LIN {X 0,Y 292.281,Z 425.223,A -85,B 0,C 180,E1 -16748.644,E2 -16748.644} C_VEL
LIN {X 0,Y 292.975,Z 416.538,A -85,B 0,C 180,E1 -16751.064,E2 -16751.064} C_VEL
LIN {X 0,Y 293.77,Z 407.489,A -85,B 0,C 180,E1 -16753.137,E2 -16753.137} C_VEL
LIN {X 0,Y 294.563,Z 398.532,A -85,B 0,C 180,E1 -16754.862,E2 -16754.862} C_VEL
LIN {X 0,Y 295.725,Z 386.736,A -85,B 0,C 180,E1 -16756.748,E2 -16756.748} C_VEL
LIN {X 0,Y 296.927,Z 373.912,A -85,B 0,C 180,E1 -16758.428,E2 -16758.428} C_VEL
LIN {X 0,Y 298.037,Z 360.895,A -85,B 0,C 180,E1 -16759.815,E2 -16759.815} C_VEL
LIN {X 0,Y 298.377,Z 356.314,A -85,B 0,C 180,E1 -16760.24,E2 -16760.24} C_VEL
LIN {X 0,Y 295.222,Z 342.197,A -85,B 0,C 180,E1 -16761.551,E2 -16761.551} C_VEL
LIN {X 0,Y 291.582,Z 327.495,A -85,B 0,C 180,E1 -16762.668,E2 -16762.668} C_VEL
LIN {X 0,Y 290.883,Z 324.481,A -85,B 0,C 180,E1 -16762.869,E2 -16762.869} C_VEL
LIN {X 0,Y 290.897,Z 319.996,A -85,B 0,C 180,E1 -16767.325,E2 -16767.325} C_VEL
LIN {X 0,Y 290.942,Z 316.936,A -85,B 0,C 180,E1 -16770.483,E2 -16770.483} C_VEL
LIN {X 0,Y 290.951,Z 314.87,A -85,B 0,C 180,E1 -16772.743,E2 -16772.743} C_VEL
LIN {X 0,Y 291.348,Z 314.866,A -85,B 0,C 180,E1 -16776.658,E2 -16776.658} C_VEL
LIN {X 0,Y 292.204,Z 318.866,A -85,B 0,C 180,E1 -16780.496,E2 -16780.496} C_VEL
LIN {X 0,Y 292.885,Z 322.76,A -85,B 0,C 180,E1 -16784.097,E2 -16784.097} C_VEL
LIN {X 0,Y 293.355,Z 325.959,A -85,B 0,C 180,E1 -16786.943,E2 -16786.943} C_VEL
LIN {X 0,Y 293.486,Z 329.298,A -85,B 0,C 180,E1 -16789.717,E2 -16789.717} C_VEL
LIN {X 0,Y 293.444,Z 333.828,A -85,B 0,C 180,E1 -16793.219,E2 -16793.219} C_VEL
LIN {X 0,Y 293.478,Z 334.871,A -85,B 0,C 180,E1 -16793.943,E2 -16793.943} C_VEL
LIN {X 0,Y 294.987,Z 338.144,A -85,B 0,C 180,E1 -16794.258,E2 -16794.258} C_VEL
LIN {X 0,Y 301.868,Z 352.507,A -85,B 0,C 180,E1 -16795.778,E2 -16795.778} C_VEL
LIN {X 0,Y 307.005,Z 365.674,A -85,B 0,C 180,E1 -16797.218,E2 -16797.218} C_VEL
LIN {X 0,Y 311.165,Z 379.228,A -85,B 0,C 180,E1 -16798.779,E2 -16798.779} C_VEL
LIN {X 0,Y 312.44,Z 384.388,A -85,B 0,C 180,E1 -16799.396,E2 -16799.396} C_VEL
LIN {X 0,Y 310.407,Z 398.606,A -85,B 0,C 180,E1 -16800.684,E2 -16800.684} C_VEL
LIN {X 0,Y 308.12,Z 411.435,A -85,B 0,C 180,E1 -16802.122,E2 -16802.122} C_VEL
LIN {X 0,Y 305.586,Z 423.472,A -85,B 0,C 180,E1 -16803.759,E2 -16803.759} C_VEL
LIN {X 0,Y 303.036,Z 435.042,A -85,B 0,C 180,E1 -16805.691,E2 -16805.691} C_VEL
LIN {X 0,Y 300.575,Z 444.936,A -85,B 0,C 180,E1 -16807.669,E2 -16807.669} C_VEL
LIN {X 0,Y 298.106,Z 454.57,A -85,B 0,C 180,E1 -16810.01,E2 -16810.01} C_VEL
LIN {X 0,Y 296.027,Z 462.55,A -85,B 0,C 180,E1 -16812.38,E2 -16812.38} C_VEL
LIN {X 0,Y 294.274,Z 469.141,A -85,B 0,C 180,E1 -16814.769,E2 -16814.769} C_VEL
LIN {X 0,Y 292.752,Z 475.226,A -85,B 0,C 180,E1 -16817.522,E2 -16817.522} C_VEL
LIN {X 0,Y 291.602,Z 479.925,A -85,B 0,C 180,E1 -16820.287,E2 -16820.287} C_VEL
LIN {X 0,Y 290.787,Z 483.367,A -85,B 0,C 180,E1 -16823.059,E2 -16823.059} C_VEL
LIN {X 0,Y 290.549,Z 485.611,A -85,B 0,C 180,E1 -16825.838,E2 -16825.838} C_VEL
LIN {X 0,Y 290.207,Z 486.77,A -85,B 0,C 180,E1 -16828.612,E2 -16828.612} C_VEL
LIN {X 0,Y 290.206,Z 486.781,A -85,B 0,C 180,E1 -16831.387,E2 -16831.387} C_VEL
LIN {X 0,Y 290.537,Z 485.67,A -85,B 0,C 180,E1 -16834.161,E2 -16834.161} C_VEL
LIN {X 0,Y 290.788,Z 483.475,A -85,B 0,C 180,E1 -16836.941,E2 -16836.941} C_VEL
LIN {X 0,Y 291.6,Z 480.092,A -85,B 0,C 180,E1 -16839.713,E2 -16839.713} C_VEL
LIN {X 0,Y 292.696,Z 475.454,A -85,B 0,C 180,E1 -16842.48,E2 -16842.48} C_VEL
LIN {X 0,Y 294.228,Z 469.42,A -85,B 0,C 180,E1 -16845.233,E2 -16845.233} C_VEL
LIN {X 0,Y 296.21,Z 461.815,A -85,B 0,C 180,E1 -16847.965,E2 -16847.965} C_VEL
LIN {X 0,Y 298.328,Z 453.69,A -85,B 0,C 180,E1 -16850.333,E2 -16850.333} C_VEL
LIN {X 0,Y 300.921,Z 443.864,A -85,B 0,C 180,E1 -16852.666,E2 -16852.666} C_VEL
LIN {X 0,Y 303.325,Z 433.821,A -85,B 0,C 180,E1 -16854.649,E2 -16854.649} C_VEL
LIN {X 0,Y 305.509,Z 423.937,A -85,B 0,C 180,E1 -16856.284,E2 -16856.284} C_VEL
LIN {X 0,Y 308.026,Z 412.234,A -85,B 0,C 180,E1 -16857.887,E2 -16857.887} C_VEL
LIN {X 0,Y 310.294,Z 399.568,A -85,B 0,C 180,E1 -16859.327,E2 -16859.327} C_VEL
LIN {X 0,Y 312.269,Z 386.595,A -85,B 0,C 180,E1 -16860.523,E2 -16860.523} C_VEL
LIN {X 0,Y 312.394,Z 384.092,A -85,B 0,C 180,E1 -16860.756,E2 -16860.756} C_VEL
LIN {X 0,Y 309.143,Z 372.05,A -85,B 0,C 180,E1 -16862.176,E2 -16862.176} C_VEL
LIN {X 0,Y 304.924,Z 359.837,A -85,B 0,C 180,E1 -16863.543,E2 -16863.543} C_VEL
LIN {X 0,Y 299.653,Z 347.585,A -85,B 0,C 180,E1 -16864.877,E2 -16864.877} C_VEL
LIN {X 0,Y 294.712,Z 337.725,A -85,B 0,C 180,E1 -16865.919,E2 -16865.919} C_VEL
LIN {X 0,Y 293.448,Z 334.746,A -85,B 0,C 180,E1 -16866.235,E2 -16866.235} C_VEL
LIN {X 0,Y 293.518,Z 331.711,A -85,B 0,C 180,E1 -16868.502,E2 -16868.502} C_VEL
LIN {X 0,Y 293.456,Z 327.245,A -85,B 0,C 180,E1 -16872.111,E2 -16872.111} C_VEL
LIN {X 0,Y 293.062,Z 323.956,A -85,B 0,C 180,E1 -16874.978,E2 -16874.978} C_VEL
LIN {X 0,Y 292.466,Z 320.438,A -85,B 0,C 180,E1 -16878.153,E2 -16878.153} C_VEL
LIN {X 0,Y 291.873,Z 317.195,A -85,B 0,C 180,E1 -16881.24,E2 -16881.24} C_VEL
LIN {X 0,Y 291.381,Z 314.808,A -85,B 0,C 180,E1 -16883.777,E2 -16883.777} C_VEL
LIN {X 0,Y 291.366,Z 314.817,A -85,B 0,C 180,E1 -16887.95,E2 -16887.95} C_VEL
LIN {X 0,Y 291.343,Z 314.814,A -85,B 0,C 180,E1 -16891.154,E2 -16891.154} C_VEL
LIN {X 0,Y 291.359,Z 314.803,A -85,B 0,C 180,E1 -16894.266,E2 -16894.266} C_VEL
LIN {X 0,Y 291.369,Z 314.804,A -85,B 0,C 180,E1 -16897.298,E2 -16897.298} C_VEL
LIN {X 0,Y 291.458,Z 314.804,A -85,B 0,C 180,E1 -16900.27,E2 -16900.27} C_VEL
LIN {X 0,Y 291.497,Z 314.792,A -85,B 0,C 180,E1 -16904.665,E2 -16904.665} C_VEL
LIN {X 0,Y 291.485,Z 314.795,A -85,B 0,C 180,E1 -16905.318,E2 -16905.318} C_VEL
LIN {X 0,Y 290.843,Z 314.882,A -85,B 0,C 180,E1 -16906.471,E2 -16906.471} C_VEL
LIN {X 0,Y 288.049,Z 315.231,A -85,B 0,C 180,E1 -16908.35,E2 -16908.35} C_VEL
LIN {X 0,Y 285.681,Z 315.524,A -85,B 0,C 180,E1 -16909.876,E2 -16909.876} C_VEL
LIN {X 0,Y 284.681,Z 315.65,A -85,B 0,C 180,E1 -16911.056,E2 -16911.056} C_VEL
LIN {X 0,Y 284.608,Z 315.659,A -85,B 0,C 180,E1 -16911.456,E2 -16911.456} C_VEL
LIN {X 0,Y 284.574,Z 315.639,A -85,B 0,C 180,E1 -16914.331,E2 -16914.331} C_VEL
LIN {X 0,Y 284.855,Z 315.608,A -85,B 0,C 180,E1 -16918.586,E2 -16918.586} C_VEL
LIN {X 0,Y 284.851,Z 315.619,A -85,B 0,C 180,E1 -16921.414,E2 -16921.414} C_VEL
LIN {X 0,Y 284.658,Z 315.643,A -85,B 0,C 180,E1 -16927.091,E2 -16927.091} C_VEL
LIN {X 0,Y 284.514,Z 315.651,A -85,B 0,C 180,E1 -16929.957,E2 -16929.957} C_VEL
LIN {X 0,Y 284.482,Z 315.673,A -85,B 0,C 180,E1 -16934.303,E2 -16934.303} C_VEL
LIN {X 0,Y 284.425,Z 315.661,A -85,B 0,C 180,E1 -16937.248,E2 -16937.248} C_VEL
LIN {X 0,Y 284.376,Z 315.677,A -85,B 0,C 180,E1 -16940.242,E2 -16940.242} C_VEL
LIN {X 0,Y 284.323,Z 315.694,A -85,B 0,C 180,E1 -16943.854,E2 -16943.854} C_VEL
LIN {X 0,Y 284.283,Z 315.69,A -85,B 0,C 180,E1 -16948.016,E2 -16948.016} C_VEL
LIN {X 0,Y 284.284,Z 315.698,A -85,B 0,C 180,E1 -16951.276,E2 -16951.276} C_VEL
LIN {X 0,Y 284.328,Z 315.807,A -85,B 0,C 180,E1 -16952.243,E2 -16952.243} C_VEL
LIN {X 0,Y 285.91,Z 322.892,A -85,B 0,C 180,E1 -16956.153,E2 -16956.153} C_VEL
LIN {X 0,Y 287.665,Z 330.708,A -85,B 0,C 180,E1 -16960.158,E2 -16960.158} C_VEL
LIN {X 0,Y 289.389,Z 338.363,A -85,B 0,C 180,E1 -16963.831,E2 -16963.831} C_VEL
LIN {X 0,Y 291.295,Z 346.482,A -85,B 0,C 180,E1 -16967.504,E2 -16967.504} C_VEL
LIN {X 0,Y 293.304,Z 354.76,A -85,B 0,C 180,E1 -16970.991,E2 -16970.991} C_VEL
LIN {X 0,Y 293.898,Z 358.498,A -85,B 0,C 180,E1 -16971.839,E2 -16971.839} C_VEL
LIN {X 0,Y 293.238,Z 368.802,A -85,B 0,C 180,E1 -16973.867,E2 -16973.867} C_VEL
LIN {X 0,Y 297.903,Z 390.014,A -85,B 0,C 180,E1 -16975.176,E2 -16975.176} C_VEL
LIN {X 0,Y 300.055,Z 405.991,A -85,B 0,C 180,E1 -16976.266,E2 -16976.266} C_VEL
LIN {X 0,Y 301.158,Z 421.763,A -85,B 0,C 180,E1 -16977.538,E2 -16977.538} C_VEL
LIN {X 0,Y 301.521,Z 436.68,A -85,B 0,C 180,E1 -16978.979,E2 -16978.979} C_VEL
LIN {X 0,Y 301.025,Z 442.79,A -85,B 0,C 180,E1 -16979.594,E2 -16979.594} C_VEL
LIN {X 0,Y 298.222,Z 456.827,A -85,B 0,C 180,E1 -16981.112,E2 -16981.112} C_VEL
LIN {X 0,Y 295.429,Z 469.104,A -85,B 0,C 180,E1 -16982.746,E2 -16982.746} C_VEL
LIN {X 0,Y 292.883,Z 479.435,A -85,B 0,C 180,E1 -16984.41,E2 -16984.41} C_VEL
LIN {X 0,Y 290.393,Z 490.022,A -85,B 0,C 180,E1 -16986.464,E2 -16986.464} C_VEL
LIN {X 0,Y 288.224,Z 499.009,A -85,B 0,C 180,E1 -16988.546,E2 -16988.546} C_VEL
LIN {X 0,Y 286.145,Z 507.863,A -85,B 0,C 180,E1 -16991.008,E2 -16991.008} C_VEL
LIN {X 0,Y 284.681,Z 515.263,A -85,B 0,C 180,E1 -16993.507,E2 -16993.507} C_VEL
LIN {X 0,Y 283.458,Z 522.136,A -85,B 0,C 180,E1 -16996.377,E2 -16996.377} C_VEL
LIN {X 0,Y 282.864,Z 527.542,A -85,B 0,C 180,E1 -16999.261,E2 -16999.261} C_VEL
LIN {X 0,Y 282.743,Z 530.67,A -85,B 0,C 180,E1 -17001.423,E2 -17001.423} C_VEL
LIN {X 0,Y 282.906,Z 533.758,A -85,B 0,C 180,E1 -17004.297,E2 -17004.297} C_VEL
LIN {X 0,Y 283.058,Z 535.604,A -85,B 0,C 180,E1 -17007.154,E2 -17007.154} C_VEL
LIN {X 0,Y 283.209,Z 536.24,A -85,B 0,C 180,E1 -17010,E2 -17010} C_VEL
LIN {X 0,Y 283.107,Z 535.603,A -85,B 0,C 180,E1 -17012.846,E2 -17012.846} C_VEL
LIN {X 0,Y 282.92,Z 533.747,A -85,B 0,C 180,E1 -17015.703,E2 -17015.703} C_VEL
LIN {X 0,Y 282.783,Z 530.648,A -85,B 0,C 180,E1 -17018.576,E2 -17018.576} C_VEL
LIN {X 0,Y 282.981,Z 526.261,A -85,B 0,C 180,E1 -17021.46,E2 -17021.46} C_VEL
LIN {X 0,Y 283.73,Z 520.505,A -85,B 0,C 180,E1 -17024.342,E2 -17024.342} C_VEL
LIN {X 0,Y 285.038,Z 513.22,A -85,B 0,C 180,E1 -17027.21,E2 -17027.21} C_VEL
LIN {X 0,Y 286.735,Z 505.442,A -85,B 0,C 180,E1 -17029.696,E2 -17029.696} C_VEL
LIN {X 0,Y 288.901,Z 496.554,A -85,B 0,C 180,E1 -17032.041,E2 -17032.041} C_VEL
LIN {X 0,Y 291.219,Z 486.613,A -85,B 0,C 180,E1 -17034.222,E2 -17034.222} C_VEL
LIN {X 0,Y 292.965,Z 479.467,A -85,B 0,C 180,E1 -17035.583,E2 -17035.583} C_VEL
LIN {X 0,Y 296.814,Z 468.953,A -85,B 0,C 180,E1 -17037.882,E2 -17037.882} C_VEL
LIN {X 0,Y 301.379,Z 457.024,A -85,B 0,C 180,E1 -17040.052,E2 -17040.052} C_VEL
LIN {X 0,Y 306.225,Z 443.816,A -85,B 0,C 180,E1 -17042.055,E2 -17042.055} C_VEL
LIN {X 0,Y 309.774,Z 429.399,A -85,B 0,C 180,E1 -17044.161,E2 -17044.161} C_VEL
LIN {X 0,Y 311.396,Z 419.284,A -85,B 0,C 180,E1 -17045.66,E2 -17045.66} C_VEL
LIN {X 0,Y 312.435,Z 406.673,A -85,B 0,C 180,E1 -17047.71,E2 -17047.71} C_VEL
LIN {X 0,Y 312.742,Z 394.992,A -85,B 0,C 180,E1 -17049.86,E2 -17049.86} C_VEL
LIN {X 0,Y 312.782,Z 389.058,A -85,B 0,C 180,E1 -17051.089,E2 -17051.089} C_VEL
LIN {X 0,Y 312.133,Z 386.452,A -85,B 0,C 180,E1 -17052.01,E2 -17052.01} C_VEL
LIN {X 0,Y 310.091,Z 381.925,A -85,B 0,C 180,E1 -17054.636,E2 -17054.636} C_VEL
LIN {X 0,Y 309.135,Z 379.146,A -85,B 0,C 180,E1 -17056.998,E2 -17056.998} C_VEL
LIN {X 0,Y 308.913,Z 377.902,A -85,B 0,C 180,E1 -17058.718,E2 -17058.718} C_VEL
LIN {X 0,Y 309.154,Z 377.322,A -85,B 0,C 180,E1 -17060.618,E2 -17060.618} C_VEL
LIN {X 0,Y 309.806,Z 377.672,A -85,B 0,C 180,E1 -17062.56,E2 -17062.56} C_VEL
LIN {X 0,Y 310.718,Z 379.097,A -85,B 0,C 180,E1 -17064.516,E2 -17064.516} C_VEL
LIN {X 0,Y 312.001,Z 381.438,A -85,B 0,C 180,E1 -17066.455,E2 -17066.455} C_VEL
LIN {X 0,Y 313.816,Z 385.948,A -85,B 0,C 180,E1 -17068.997,E2 -17068.997} C_VEL
LIN {X 0,Y 315.619,Z 391.802,A -85,B 0,C 180,E1 -17071.451,E2 -17071.451} C_VEL
LIN {X 0,Y 316.372,Z 395.772,A -85,B 0,C 180,E1 -17072.838,E2 -17072.838} C_VEL
LIN {X 0,Y 311.508,Z 407.708,A -85,B 0,C 180,E1 -17074.879,E2 -17074.879} C_VEL
LIN {X 0,Y 306.8,Z 418.029,A -85,B 0,C 180,E1 -17077.081,E2 -17077.081} C_VEL
LIN {X 0,Y 302.738,Z 426.283,A -85,B 0,C 180,E1 -17079.266,E2 -17079.266} C_VEL
LIN {X 0,Y 299.02,Z 432.975,A -85,B 0,C 180,E1 -17081.501,E2 -17081.501} C_VEL
LIN {X 0,Y 295.395,Z 439.029,A -85,B 0,C 180,E1 -17084.121,E2 -17084.121} C_VEL
LIN {X 0,Y 293.012,Z 442.485,A -85,B 0,C 180,E1 -17086.122,E2 -17086.122} C_VEL
LIN {X 0,Y 290.368,Z 445.829,A -85,B 0,C 180,E1 -17088.835,E2 -17088.835} C_VEL
LIN {X 0,Y 289.19,Z 446.951,A -85,B 0,C 180,E1 -17090.206,E2 -17090.206} C_VEL
LIN {X 0,Y 287.411,Z 448.034,A -85,B 0,C 180,E1 -17092.977,E2 -17092.977} C_VEL
LIN {X 0,Y 286.208,Z 447.668,A -85,B 0,C 180,E1 -17095.776,E2 -17095.776} C_VEL
LIN {X 0,Y 285.571,Z 446.967,A -85,B 0,C 180,E1 -17097.179,E2 -17097.179} C_VEL
LIN {X 0,Y 285.274,Z 445.858,A -85,B 0,C 180,E1 -17098.588,E2 -17098.588} C_VEL
LIN {X 0,Y 284.786,Z 444.375,A -85,B 0,C 180,E1 -17100,E2 -17100} C_VEL
LIN {X 0,Y 284.572,Z 441.39,A -85,B 0,C 180,E1 -17102.123,E2 -17102.123} C_VEL
LIN {X 0,Y 284.356,Z 437.471,A -85,B 0,C 180,E1 -17104.252,E2 -17104.252} C_VEL
LIN {X 0,Y 284.781,Z 432.533,A -85,B 0,C 180,E1 -17106.376,E2 -17106.376} C_VEL
LIN {X 0,Y 285.266,Z 425.416,A -85,B 0,C 180,E1 -17108.847,E2 -17108.847} C_VEL
LIN {X 0,Y 285.982,Z 416.448,A -85,B 0,C 180,E1 -17111.338,E2 -17111.338} C_VEL
LIN {X 0,Y 286.82,Z 407.169,A -85,B 0,C 180,E1 -17113.461,E2 -17113.461} C_VEL
LIN {X 0,Y 287.803,Z 395.908,A -85,B 0,C 180,E1 -17115.582,E2 -17115.582} C_VEL
LIN {X 0,Y 289.17,Z 383.463,A -85,B 0,C 180,E1 -17117.504,E2 -17117.504} C_VEL
LIN {X 0,Y 290.389,Z 369.241,A -85,B 0,C 180,E1 -17119.285,E2 -17119.285} C_VEL
LIN {X 0,Y 291.404,Z 357.506,A -85,B 0,C 180,E1 -17120.47,E2 -17120.47} C_VEL
LIN {X 0,Y 288.49,Z 344.156,A -85,B 0,C 180,E1 -17121.754,E2 -17121.754} C_VEL
LIN {X 0,Y 284.743,Z 328.927,A -85,B 0,C 180,E1 -17122.954,E2 -17122.954} C_VEL
LIN {X 0,Y 283.856,Z 325.076,A -85,B 0,C 180,E1 -17123.23,E2 -17123.23} C_VEL
LIN {X 0,Y 283.857,Z 321.34,A -85,B 0,C 180,E1 -17126.959,E2 -17126.959} C_VEL
LIN {X 0,Y 283.927,Z 318.431,A -85,B 0,C 180,E1 -17129.962,E2 -17129.962} C_VEL
LIN {X 0,Y 283.937,Z 315.742,A -85,B 0,C 180,E1 -17132.994,E2 -17132.994} C_VEL
LIN {X 0,Y 284.182,Z 315.865,A -85,B 0,C 180,E1 -17135.47,E2 -17135.47} C_VEL
LIN {X 0,Y 284.889,Z 318.482,A -85,B 0,C 180,E1 -17138.078,E2 -17138.078} C_VEL
LIN {X 0,Y 285.626,Z 322.113,A -85,B 0,C 180,E1 -17141.633,E2 -17141.633} C_VEL
LIN {X 0,Y 286.302,Z 326.199,A -85,B 0,C 180,E1 -17145.388,E2 -17145.388} C_VEL
LIN {X 0,Y 286.676,Z 329.839,A -85,B 0,C 180,E1 -17148.553,E2 -17148.553} C_VEL
LIN {X 0,Y 286.606,Z 335.245,A -85,B 0,C 180,E1 -17152.825,E2 -17152.825} C_VEL
LIN {X 0,Y 286.734,Z 335.84,A -85,B 0,C 180,E1 -17152.967,E2 -17152.967} C_VEL
LIN {X 0,Y 288.261,Z 338.94,A -85,B 0,C 180,E1 -17153.296,E2 -17153.296} C_VEL
LIN {X 0,Y 294.647,Z 351.97,A -85,B 0,C 180,E1 -17154.758,E2 -17154.758} C_VEL
LIN {X 0,Y 299.925,Z 364.933,A -85,B 0,C 180,E1 -17156.242,E2 -17156.242} C_VEL
LIN {X 0,Y 304.193,Z 378.259,A -85,B 0,C 180,E1 -17157.83,E2 -17157.83} C_VEL
LIN {X 0,Y 306.061,Z 385.562,A -85,B 0,C 180,E1 -17158.744,E2 -17158.744} C_VEL
LIN {X 0,Y 305.672,Z 390.296,A -85,B 0,C 180,E1 -17159.176,E2 -17159.176} C_VEL
LIN {X 0,Y 303.514,Z 403.795,A -85,B 0,C 180,E1 -17160.524,E2 -17160.524} C_VEL
LIN {X 0,Y 300.819,Z 417.049,A -85,B 0,C 180,E1 -17162.143,E2 -17162.143} C_VEL
LIN {X 0,Y 298.096,Z 429.254,A -85,B 0,C 180,E1 -17163.99,E2 -17163.99} C_VEL
LIN {X 0,Y 295.348,Z 440.8,A -85,B 0,C 180,E1 -17166.138,E2 -17166.138} C_VEL
LIN {X 0,Y 292.917,Z 449.874,A -85,B 0,C 180,E1 -17168.167,E2 -17168.167} C_VEL
LIN {X 0,Y 290.461,Z 458.624,A -85,B 0,C 180,E1 -17170.523,E2 -17170.523} C_VEL
LIN {X 0,Y 288.429,Z 466.128,A -85,B 0,C 180,E1 -17172.998,E2 -17172.998} C_VEL
LIN {X 0,Y 286.576,Z 472.977,A -85,B 0,C 180,E1 -17175.804,E2 -17175.804} C_VEL
LIN {X 0,Y 285.176,Z 478.35,A -85,B 0,C 180,E1 -17178.629,E2 -17178.629} C_VEL
LIN {X 0,Y 284.114,Z 482.658,A -85,B 0,C 180,E1 -17181.676,E2 -17181.676} C_VEL
LIN {X 0,Y 283.546,Z 485.244,A -85,B 0,C 180,E1 -17184.31,E2 -17184.31} C_VEL
LIN {X 0,Y 283.505,Z 486.218,A -85,B 0,C 180,E1 -17185.735,E2 -17185.735} C_VEL
LIN {X 0,Y 283.149,Z 487.377,A -85,B 0,C 180,E1 -17188.577,E2 -17188.577} C_VEL
LIN {X 0,Y 283.148,Z 487.388,A -85,B 0,C 180,E1 -17191.422,E2 -17191.422} C_VEL
LIN {X 0,Y 283.494,Z 486.277,A -85,B 0,C 180,E1 -17194.265,E2 -17194.265} C_VEL
LIN {X 0,Y 283.774,Z 484.082,A -85,B 0,C 180,E1 -17197.113,E2 -17197.113} C_VEL
LIN {X 0,Y 284.634,Z 480.698,A -85,B 0,C 180,E1 -17199.953,E2 -17199.953} C_VEL
LIN {X 0,Y 285.778,Z 476.062,A -85,B 0,C 180,E1 -17202.787,E2 -17202.787} C_VEL
LIN {X 0,Y 287.381,Z 470.028,A -85,B 0,C 180,E1 -17205.605,E2 -17205.605} C_VEL
LIN {X 0,Y 289.474,Z 462.421,A -85,B 0,C 180,E1 -17208.398,E2 -17208.398} C_VEL
LIN {X 0,Y 291.697,Z 454.293,A -85,B 0,C 180,E1 -17210.816,E2 -17210.816} C_VEL
LIN {X 0,Y 294.402,Z 444.464,A -85,B 0,C 180,E1 -17213.196,E2 -17213.196} C_VEL
LIN {X 0,Y 296.902,Z 434.419,A -85,B 0,C 180,E1 -17215.219,E2 -17215.219} C_VEL
LIN {X 0,Y 299.181,Z 424.533,A -85,B 0,C 180,E1 -17216.884,E2 -17216.884} C_VEL
LIN {X 0,Y 302.054,Z 411.57,A -85,B 0,C 180,E1 -17218.678,E2 -17218.678} C_VEL
LIN {X 0,Y 304.425,Z 398.618,A -85,B 0,C 180,E1 -17220.14,E2 -17220.14} C_VEL
LIN {X 0,Y 306.217,Z 386.977,A -85,B 0,C 180,E1 -17221.213,E2 -17221.213} C_VEL
LIN {X 0,Y 304.343,Z 378.729,A -85,B 0,C 180,E1 -17222.23,E2 -17222.23} C_VEL
LIN {X 0,Y 300.361,Z 366.023,A -85,B 0,C 180,E1 -17223.747,E2 -17223.747} C_VEL
LIN {X 0,Y 295.504,Z 353.884,A -85,B 0,C 180,E1 -17225.153,E2 -17225.153} C_VEL
LIN {X 0,Y 289.995,Z 342.297,A -85,B 0,C 180,E1 -17226.457,E2 -17226.457} C_VEL
LIN {X 0,Y 286.814,Z 336.104,A -85,B 0,C 180,E1 -17227.141,E2 -17227.141} C_VEL
LIN {X 0,Y 286.611,Z 335.375,A -85,B 0,C 180,E1 -17227.225,E2 -17227.225} C_VEL
LIN {X 0,Y 286.641,Z 331.154,A -85,B 0,C 180,E1 -17230.529,E2 -17230.529} C_VEL
LIN {X 0,Y 286.502,Z 327.733,A -85,B 0,C 180,E1 -17233.381,E2 -17233.381} C_VEL
LIN {X 0,Y 285.797,Z 323.189,A -85,B 0,C 180,E1 -17237.538,E2 -17237.538} C_VEL
LIN {X 0,Y 285.323,Z 320.478,A -85,B 0,C 180,E1 -17240.176,E2 -17240.176} C_VEL
LIN {X 0,Y 284.62,Z 316.929,A -85,B 0,C 180,E1 -17243.656,E2 -17243.656} C_VEL
LIN {X 0,Y 284.343,Z 315.694,A -85,B 0,C 180,E1 -17244.999,E2 -17244.999} C_VEL
LIN {X 0,Y 284.285,Z 315.694,A -85,B 0,C 180,E1 -17248.724,E2 -17248.724} C_VEL
LIN {X 0,Y 284.282,Z 315.7,A -85,B 0,C 180,E1 -17251.984,E2 -17251.984} C_VEL
LIN {X 0,Y 284.323,Z 315.695,A -85,B 0,C 180,E1 -17256.145,E2 -17256.145} C_VEL
LIN {X 0,Y 284.376,Z 315.682,A -85,B 0,C 180,E1 -17259.904,E2 -17259.904} C_VEL
LIN {X 0,Y 284.447,Z 315.667,A -85,B 0,C 180,E1 -17264.492,E2 -17264.492} C_VEL
LIN {X 0,Y 284.482,Z 315.651,A -85,B 0,C 180,E1 -17268.601,E2 -17268.601} C_VEL
LIN {X 0,Y 284.608,Z 315.659,A -85,B 0,C 180,E1 -17271.456,E2 -17271.456} C_VEL
LIN {X 0,Y 283.962,Z 315.743,A -85,B 0,C 180,E1 -17272.636,E2 -17272.636} C_VEL
LIN {X 0,Y 281.129,Z 316.101,A -85,B 0,C 180,E1 -17274.558,E2 -17274.558} C_VEL
LIN {X 0,Y 278.749,Z 316.393,A -85,B 0,C 180,E1 -17276.119,E2 -17276.119} C_VEL
LIN {X 0,Y 277.779,Z 316.507,A -85,B 0,C 180,E1 -17277.329,E2 -17277.329} C_VEL
LIN {X 0,Y 277.728,Z 316.504,A -85,B 0,C 180,E1 -17277.738,E2 -17277.738} C_VEL
LIN {X 0,Y 277.872,Z 316.472,A -85,B 0,C 180,E1 -17280,E2 -17280} C_VEL
LIN {X 0,Y 277.685,Z 316.521,A -85,B 0,C 180,E1 -17282.901,E2 -17282.901} C_VEL
LIN {X 0,Y 277.615,Z 316.522,A -85,B 0,C 180,E1 -17287.272,E2 -17287.272} C_VEL
LIN {X 0,Y 277.457,Z 316.527,A -85,B 0,C 180,E1 -17290.213,E2 -17290.213} C_VEL
LIN {X 0,Y 277.435,Z 316.544,A -85,B 0,C 180,E1 -17294.674,E2 -17294.674} C_VEL
LIN {X 0,Y 277.345,Z 316.564,A -85,B 0,C 180,E1 -17299.234,E2 -17299.234} C_VEL
LIN {X 0,Y 277.279,Z 316.573,A -85,B 0,C 180,E1 -17304.152,E2 -17304.152} C_VEL
LIN {X 0,Y 277.269,Z 316.557,A -85,B 0,C 180,E1 -17307.483,E2 -17307.483} C_VEL
LIN {X 0,Y 277.277,Z 316.626,A -85,B 0,C 180,E1 -17311.518,E2 -17311.518} C_VEL
LIN {X 0,Y 278.781,Z 323.501,A -85,B 0,C 180,E1 -17315.438,E2 -17315.438} C_VEL
LIN {X 0,Y 280.611,Z 331.528,A -85,B 0,C 180,E1 -17319.691,E2 -17319.691} C_VEL
LIN {X 0,Y 282.614,Z 340.564,A -85,B 0,C 180,E1 -17324.131,E2 -17324.131} C_VEL
LIN {X 0,Y 284.495,Z 348.537,A -85,B 0,C 180,E1 -17327.825,E2 -17327.825} C_VEL
LIN {X 0,Y 285.12,Z 350.958,A -85,B 0,C 180,E1 -17328.871,E2 -17328.871} C_VEL
LIN {X 0,Y 287.39,Z 359.286,A -85,B 0,C 180,E1 -17331.047,E2 -17331.047} C_VEL
LIN {X 0,Y 287.427,Z 363.003,A -85,B 0,C 180,E1 -17331.858,E2 -17331.858} C_VEL
LIN {X 0,Y 286.926,Z 368.206,A -85,B 0,C 180,E1 -17332.925,E2 -17332.925} C_VEL
LIN {X 0,Y 291.899,Z 390.588,A -85,B 0,C 180,E1 -17334.404,E2 -17334.404} C_VEL
LIN {X 0,Y 293.918,Z 406.526,A -85,B 0,C 180,E1 -17335.54,E2 -17335.54} C_VEL
LIN {X 0,Y 294.815,Z 421.152,A -85,B 0,C 180,E1 -17336.751,E2 -17336.751} C_VEL
LIN {X 0,Y 295.148,Z 436.187,A -85,B 0,C 180,E1 -17338.245,E2 -17338.245} C_VEL
LIN {X 0,Y 294.694,Z 443.103,A -85,B 0,C 180,E1 -17338.983,E2 -17338.983} C_VEL
LIN {X 0,Y 291.968,Z 456.228,A -85,B 0,C 180,E1 -17340.432,E2 -17340.432} C_VEL
LIN {X 0,Y 289.051,Z 468.498,A -85,B 0,C 180,E1 -17342.093,E2 -17342.093} C_VEL
LIN {X 0,Y 286.435,Z 478.83,A -85,B 0,C 180,E1 -17343.791,E2 -17343.791} C_VEL
LIN {X 0,Y 283.798,Z 489.41,A -85,B 0,C 180,E1 -17345.883,E2 -17345.883} C_VEL
LIN {X 0,Y 281.177,Z 499.77,A -85,B 0,C 180,E1 -17348.366,E2 -17348.366} C_VEL
LIN {X 0,Y 279.06,Z 508.386,A -85,B 0,C 180,E1 -17350.889,E2 -17350.889} C_VEL
LIN {X 0,Y 277.394,Z 516.505,A -85,B 0,C 180,E1 -17353.818,E2 -17353.818} C_VEL
LIN {X 0,Y 276.246,Z 522.992,A -85,B 0,C 180,E1 -17356.764,E2 -17356.764} C_VEL
LIN {X 0,Y 275.729,Z 528.036,A -85,B 0,C 180,E1 -17359.722,E2 -17359.722} C_VEL
LIN {X 0,Y 275.701,Z 531.756,A -85,B 0,C 180,E1 -17362.678,E2 -17362.678} C_VEL
LIN {X 0,Y 275.832,Z 533.147,A -85,B 0,C 180,E1 -17364.151,E2 -17364.151} C_VEL
LIN {X 0,Y 275.963,Z 534.993,A -85,B 0,C 180,E1 -17367.081,E2 -17367.081} C_VEL
LIN {X 0,Y 276.093,Z 535.469,A -85,B 0,C 180,E1 -17368.542,E2 -17368.542} C_VEL
LIN {X 0,Y 276.143,Z 535.633,A -85,B 0,C 180,E1 -17370,E2 -17370} C_VEL
LIN {X 0,Y 276.01,Z 534.992,A -85,B 0,C 180,E1 -17372.919,E2 -17372.919} C_VEL
LIN {X 0,Y 275.814,Z 532.68,A -85,B 0,C 180,E1 -17376.407,E2 -17376.407} C_VEL
LIN {X 0,Y 275.72,Z 529.092,A -85,B 0,C 180,E1 -17379.537,E2 -17379.537} C_VEL
LIN {X 0,Y 276.12,Z 524.357,A -85,B 0,C 180,E1 -17382.495,E2 -17382.495} C_VEL
LIN {X 0,Y 277.016,Z 518.322,A -85,B 0,C 180,E1 -17385.405,E2 -17385.405} C_VEL
LIN {X 0,Y 278.566,Z 510.531,A -85,B 0,C 180,E1 -17388.383,E2 -17388.383} C_VEL
LIN {X 0,Y 280.606,Z 502.317,A -85,B 0,C 180,E1 -17390.91,E2 -17390.91} C_VEL
LIN {X 0,Y 283.002,Z 492.465,A -85,B 0,C 180,E1 -17393.412,E2 -17393.412} C_VEL
LIN {X 0,Y 285.548,Z 482.494,A -85,B 0,C 180,E1 -17395.513,E2 -17395.513} C_VEL
LIN {X 0,Y 289.975,Z 471.309,A -85,B 0,C 180,E1 -17398.205,E2 -17398.205} C_VEL
LIN {X 0,Y 295.424,Z 458.079,A -85,B 0,C 180,E1 -17400.763,E2 -17400.763} C_VEL
LIN {X 0,Y 300.415,Z 445.598,A -85,B 0,C 180,E1 -17402.752,E2 -17402.752} C_VEL
LIN {X 0,Y 304.302,Z 431.965,A -85,B 0,C 180,E1 -17404.863,E2 -17404.863} C_VEL
LIN {X 0,Y 306.258,Z 422.529,A -85,B 0,C 180,E1 -17406.353,E2 -17406.353} C_VEL
LIN {X 0,Y 307.74,Z 410.784,A -85,B 0,C 180,E1 -17408.349,E2 -17408.349} C_VEL
LIN {X 0,Y 308.684,Z 398.969,A -85,B 0,C 180,E1 -17410.645,E2 -17410.645} C_VEL
LIN {X 0,Y 308.934,Z 394.037,A -85,B 0,C 180,E1 -17411.714,E2 -17411.714} C_VEL
LIN {X 0,Y 308.68,Z 392.72,A -85,B 0,C 180,E1 -17412.2,E2 -17412.2} C_VEL
LIN {X 0,Y 307.271,Z 389.29,A -85,B 0,C 180,E1 -17414.101,E2 -17414.101} C_VEL
LIN {X 0,Y 306.209,Z 386.119,A -85,B 0,C 180,E1 -17416.485,E2 -17416.485} C_VEL
LIN {X 0,Y 305.812,Z 384.089,A -85,B 0,C 180,E1 -17419.323,E2 -17419.323} C_VEL
LIN {X 0,Y 306.202,Z 383.736,A -85,B 0,C 180,E1 -17421.705,E2 -17421.705} C_VEL
LIN {X 0,Y 306.812,Z 384.516,A -85,B 0,C 180,E1 -17423.447,E2 -17423.447} C_VEL
LIN {X 0,Y 308.086,Z 387.118,A -85,B 0,C 180,E1 -17426.102,E2 -17426.102} C_VEL
LIN {X 0,Y 309.454,Z 391.026,A -85,B 0,C 180,E1 -17428.51,E2 -17428.51} C_VEL
LIN {X 0,Y 310.778,Z 396.356,A -85,B 0,C 180,E1 -17430.964,E2 -17430.964} C_VEL
LIN {X 0,Y 311.134,Z 398.401,A -85,B 0,C 180,E1 -17431.758,E2 -17431.758} C_VEL
LIN {X 0,Y 311.001,Z 400.34,A -85,B 0,C 180,E1 -17432.329,E2 -17432.329} C_VEL
LIN {X 0,Y 306.318,Z 410.593,A -85,B 0,C 180,E1 -17434.156,E2 -17434.156} C_VEL
LIN {X 0,Y 301.513,Z 420.203,A -85,B 0,C 180,E1 -17436.292,E2 -17436.292} C_VEL
LIN {X 0,Y 297.187,Z 428.2,A -85,B 0,C 180,E1 -17438.497,E2 -17438.497} C_VEL
LIN {X 0,Y 292.718,Z 435.594,A -85,B 0,C 180,E1 -17441.087,E2 -17441.087} C_VEL
LIN {X 0,Y 288.902,Z 441.288,A -85,B 0,C 180,E1 -17443.755,E2 -17443.755} C_VEL
LIN {X 0,Y 286.433,Z 444.53,A -85,B 0,C 180,E1 -17445.797,E2 -17445.797} C_VEL
LIN {X 0,Y 283.62,Z 447.558,A -85,B 0,C 180,E1 -17448.566,E2 -17448.566} C_VEL
LIN {X 0,Y 281.369,Z 449.145,A -85,B 0,C 180,E1 -17451.381,E2 -17451.381} C_VEL
LIN {X 0,Y 279.821,Z 449.273,A -85,B 0,C 180,E1 -17454.234,E2 -17454.234} C_VEL
LIN {X 0,Y 279.229,Z 448.814,A -85,B 0,C 180,E1 -17455.67,E2 -17455.67} C_VEL
LIN {X 0,Y 278.566,Z 447.994,A -85,B 0,C 180,E1 -17457.108,E2 -17457.108} C_VEL
LIN {X 0,Y 278.255,Z 446.744,A -85,B 0,C 180,E1 -17458.553,E2 -17458.553} C_VEL
LIN {X 0,Y 277.684,Z 444.229,A -85,B 0,C 180,E1 -17460.725,E2 -17460.725} C_VEL
LIN {X 0,Y 277.381,Z 440.772,A -85,B 0,C 180,E1 -17462.905,E2 -17462.905} C_VEL
LIN {X 0,Y 277.455,Z 436.333,A -85,B 0,C 180,E1 -17465.086,E2 -17465.086} C_VEL
LIN {X 0,Y 277.939,Z 429.861,A -85,B 0,C 180,E1 -17467.629,E2 -17467.629} C_VEL
LIN {X 0,Y 278.537,Z 421.504,A -85,B 0,C 180,E1 -17470.247,E2 -17470.247} C_VEL
LIN {X 0,Y 279.247,Z 413.322,A -85,B 0,C 180,E1 -17472.353,E2 -17472.353} C_VEL
LIN {X 0,Y 280.156,Z 403.167,A -85,B 0,C 180,E1 -17474.529,E2 -17474.529} C_VEL
LIN {X 0,Y 281.43,Z 390.835,A -85,B 0,C 180,E1 -17476.69,E2 -17476.69} C_VEL
LIN {X 0,Y 282.662,Z 378.353,A -85,B 0,C 180,E1 -17478.482,E2 -17478.482} C_VEL
LIN {X 0,Y 283.968,Z 364.057,A -85,B 0,C 180,E1 -17480.15,E2 -17480.15} C_VEL
LIN {X 0,Y 284.374,Z 357.804,A -85,B 0,C 180,E1 -17480.772,E2 -17480.772} C_VEL
LIN {X 0,Y 280.925,Z 342.8,A -85,B 0,C 180,E1 -17482.233,E2 -17482.233} C_VEL
LIN {X 0,Y 277.287,Z 327.78,A -85,B 0,C 180,E1 -17483.41,E2 -17483.41} C_VEL
LIN {X 0,Y 276.821,Z 325.692,A -85,B 0,C 180,E1 -17483.566,E2 -17483.566} C_VEL
LIN {X 0,Y 276.841,Z 321.982,A -85,B 0,C 180,E1 -17487.311,E2 -17487.311} C_VEL
LIN {X 0,Y 276.884,Z 318.925,A -85,B 0,C 180,E1 -17490.508,E2 -17490.508} C_VEL
LIN {X 0,Y 276.894,Z 316.617,A -85,B 0,C 180,E1 -17493.113,E2 -17493.113} C_VEL
LIN {X 0,Y 276.984,Z 316.706,A -85,B 0,C 180,E1 -17493.932,E2 -17493.932} C_VEL
LIN {X 0,Y 277.953,Z 319.947,A -85,B 0,C 180,E1 -17497.361,E2 -17497.361} C_VEL
LIN {X 0,Y 278.721,Z 323.564,A -85,B 0,C 180,E1 -17500.965,E2 -17500.965} C_VEL
LIN {X 0,Y 279.492,Z 328.09,A -85,B 0,C 180,E1 -17505.244,E2 -17505.244} C_VEL
LIN {X 0,Y 279.784,Z 330.398,A -85,B 0,C 180,E1 -17507.295,E2 -17507.295} C_VEL
LIN {X 0,Y 279.835,Z 333.88,A -85,B 0,C 180,E1 -17510.176,E2 -17510.176} C_VEL
LIN {X 0,Y 279.886,Z 336.179,A -85,B 0,C 180,E1 -17511.893,E2 -17511.893} C_VEL
LIN {X 0,Y 281.481,Z 339.551,A -85,B 0,C 180,E1 -17512.26,E2 -17512.26} C_VEL
LIN {X 0,Y 287.749,Z 352.113,A -85,B 0,C 180,E1 -17513.755,E2 -17513.755} C_VEL
LIN {X 0,Y 293.214,Z 365.239,A -85,B 0,C 180,E1 -17515.336,E2 -17515.336} C_VEL
LIN {X 0,Y 297.207,Z 377.357,A -85,B 0,C 180,E1 -17516.832,E2 -17516.832} C_VEL
LIN {X 0,Y 299.98,Z 388.263,A -85,B 0,C 180,E1 -17518.256,E2 -17518.256} C_VEL
LIN {X 0,Y 297.919,Z 401.326,A -85,B 0,C 180,E1 -17519.523,E2 -17519.523} C_VEL
LIN {X 0,Y 295.159,Z 415.141,A -85,B 0,C 180,E1 -17521.172,E2 -17521.172} C_VEL
LIN {X 0,Y 292.498,Z 426.547,A -85,B 0,C 180,E1 -17522.837,E2 -17522.837} C_VEL
LIN {X 0,Y 289.775,Z 437.979,A -85,B 0,C 180,E1 -17524.885,E2 -17524.885} C_VEL
LIN {X 0,Y 287.118,Z 447.601,A -85,B 0,C 180,E1 -17526.943,E2 -17526.943} C_VEL
LIN {X 0,Y 284.46,Z 456.987,A -85,B 0,C 180,E1 -17529.386,E2 -17529.386} C_VEL
LIN {X 0,Y 282.271,Z 464.783,A -85,B 0,C 180,E1 -17531.867,E2 -17531.867} C_VEL
LIN {X 0,Y 280.159,Z 472.031,A -85,B 0,C 180,E1 -17534.728,E2 -17534.728} C_VEL
LIN {X 0,Y 278.595,Z 477.761,A -85,B 0,C 180,E1 -17537.618,E2 -17537.618} C_VEL
LIN {X 0,Y 277.656,Z 481.144,A -85,B 0,C 180,E1 -17539.794,E2 -17539.794} C_VEL
LIN {X 0,Y 276.76,Z 484.583,A -85,B 0,C 180,E1 -17542.705,E2 -17542.705} C_VEL
LIN {X 0,Y 276.462,Z 486.826,A -85,B 0,C 180,E1 -17545.626,E2 -17545.626} C_VEL
LIN {X 0,Y 276.094,Z 487.984,A -85,B 0,C 180,E1 -17548.541,E2 -17548.541} C_VEL
LIN {X 0,Y 276.093,Z 487.995,A -85,B 0,C 180,E1 -17551.458,E2 -17551.458} C_VEL
LIN {X 0,Y 276.451,Z 486.884,A -85,B 0,C 180,E1 -17554.374,E2 -17554.374} C_VEL
LIN {X 0,Y 276.764,Z 484.689,A -85,B 0,C 180,E1 -17557.294,E2 -17557.294} C_VEL
LIN {X 0,Y 277.652,Z 481.307,A -85,B 0,C 180,E1 -17560.206,E2 -17560.206} C_VEL
LIN {X 0,Y 278.873,Z 476.669,A -85,B 0,C 180,E1 -17563.109,E2 -17563.109} C_VEL
LIN {X 0,Y 280.55,Z 470.635,A -85,B 0,C 180,E1 -17565.995,E2 -17565.995} C_VEL
LIN {X 0,Y 282.755,Z 463.026,A -85,B 0,C 180,E1 -17568.851,E2 -17568.851} C_VEL
LIN {X 0,Y 285.1,Z 454.895,A -85,B 0,C 180,E1 -17571.321,E2 -17571.321} C_VEL
LIN {X 0,Y 287.913,Z 445.064,A -85,B 0,C 180,E1 -17573.751,E2 -17573.751} C_VEL
LIN {X 0,Y 290.507,Z 435.018,A -85,B 0,C 180,E1 -17575.814,E2 -17575.814} C_VEL
LIN {X 0,Y 293.182,Z 424.079,A -85,B 0,C 180,E1 -17577.673,E2 -17577.673} C_VEL
LIN {X 0,Y 296.112,Z 410.847,A -85,B 0,C 180,E1 -17579.504,E2 -17579.504} C_VEL
LIN {X 0,Y 298.662,Z 397.598,A -85,B 0,C 180,E1 -17580.981,E2 -17580.981} C_VEL
LIN {X 0,Y 300.04,Z 388.603,A -85,B 0,C 180,E1 -17581.822,E2 -17581.822} C_VEL
LIN {X 0,Y 297.464,Z 377.983,A -85,B 0,C 180,E1 -17583.201,E2 -17583.201} C_VEL
LIN {X 0,Y 293.313,Z 365.35,A -85,B 0,C 180,E1 -17584.769,E2 -17584.769} C_VEL
LIN {X 0,Y 287.9,Z 352.437,A -85,B 0,C 180,E1 -17586.334,E2 -17586.334} C_VEL
LIN {X 0,Y 283.31,Z 343.044,A -85,B 0,C 180,E1 -17587.456,E2 -17587.456} C_VEL
LIN {X 0,Y 280.938,Z 338.728,A -85,B 0,C 180,E1 -17587.985,E2 -17587.985} C_VEL
LIN {X 0,Y 279.845,Z 336.006,A -85,B 0,C 180,E1 -17588.29,E2 -17588.29} C_VEL
LIN {X 0,Y 279.821,Z 332.49,A -85,B 0,C 180,E1 -17591.107,E2 -17591.107} C_VEL
LIN {X 0,Y 279.738,Z 329.952,A -85,B 0,C 180,E1 -17593.232,E2 -17593.232} C_VEL
LIN {X 0,Y 279.075,Z 325.693,A -85,B 0,C 180,E1 -17597.16,E2 -17597.16} C_VEL
LIN {X 0,Y 278.402,Z 321.963,A -85,B 0,C 180,E1 -17600.868,E2 -17600.868} C_VEL
LIN {X 0,Y 277.68,Z 318.371,A -85,B 0,C 180,E1 -17604.4,E2 -17604.4} C_VEL
LIN {X 0,Y 277.236,Z 316.566,A -85,B 0,C 180,E1 -17606.322,E2 -17606.322} C_VEL
LIN {X 0,Y 277.261,Z 316.561,A -85,B 0,C 180,E1 -17609.538,E2 -17609.538} C_VEL
LIN {X 0,Y 277.291,Z 316.56,A -85,B 0,C 180,E1 -17612.857,E2 -17612.857} C_VEL
LIN {X 0,Y 277.284,Z 316.572,A -85,B 0,C 180,E1 -17616.075,E2 -17616.075} C_VEL
LIN {X 0,Y 277.329,Z 316.566,A -85,B 0,C 180,E1 -17620.765,E2 -17620.765} C_VEL
LIN {X 0,Y 277.41,Z 316.554,A -85,B 0,C 180,E1 -17625.324,E2 -17625.324} C_VEL
LIN {X 0,Y 277.457,Z 316.536,A -85,B 0,C 180,E1 -17629.787,E2 -17629.787} C_VEL
LIN {X 0,Y 277.601,Z 316.514,A -85,B 0,C 180,E1 -17632.728,E2 -17632.728} C_VEL
LIN {X 0,Y 277.728,Z 316.504,A -85,B 0,C 180,E1 -17637.738,E2 -17637.738} C_VEL
LIN {X 0,Y 277.126,Z 316.569,A -85,B 0,C 180,E1 -17638.95,E2 -17638.95} C_VEL
LIN {X 0,Y 274.244,Z 316.931,A -85,B 0,C 180,E1 -17640.921,E2 -17640.921} C_VEL
LIN {X 0,Y 271.705,Z 317.266,A -85,B 0,C 180,E1 -17642.523,E2 -17642.523} C_VEL
LIN {X 0,Y 270.549,Z 317.396,A -85,B 0,C 180,E1 -17643.766,E2 -17643.766} C_VEL
LIN {X 0,Y 270.423,Z 317.405,A -85,B 0,C 180,E1 -17644.189,E2 -17644.189} C_VEL
LIN {X 0,Y 270.574,Z 317.401,A -85,B 0,C 180,E1 -17647.462,E2 -17647.462} C_VEL
LIN {X 0,Y 270.41,Z 317.402,A -85,B 0,C 180,E1 -17650.482,E2 -17650.482} C_VEL
LIN {X 0,Y 270.403,Z 317.413,A -85,B 0,C 180,E1 -17655.064,E2 -17655.064} C_VEL
LIN {X 0,Y 270.301,Z 317.437,A -85,B 0,C 180,E1 -17659.755,E2 -17659.755} C_VEL
LIN {X 0,Y 270.224,Z 317.449,A -85,B 0,C 180,E1 -17664.59,E2 -17664.59} C_VEL
LIN {X 0,Y 270.198,Z 317.442,A -85,B 0,C 180,E1 -17667.917,E2 -17667.917} C_VEL
LIN {X 0,Y 270.232,Z 317.635,A -85,B 0,C 180,E1 -17670.881,E2 -17670.881} C_VEL
LIN {X 0,Y 271.688,Z 324.044,A -85,B 0,C 180,E1 -17674.687,E2 -17674.687} C_VEL
LIN {X 0,Y 273.376,Z 331.692,A -85,B 0,C 180,E1 -17678.878,E2 -17678.878} C_VEL
LIN {X 0,Y 275.035,Z 339.202,A -85,B 0,C 180,E1 -17682.731,E2 -17682.731} C_VEL
LIN {X 0,Y 276.801,Z 346.705,A -85,B 0,C 180,E1 -17686.354,E2 -17686.354} C_VEL
LIN {X 0,Y 279.779,Z 357.452,A -85,B 0,C 180,E1 -17689.452,E2 -17689.452} C_VEL
LIN {X 0,Y 281.103,Z 362.432,A -85,B 0,C 180,E1 -17690.809,E2 -17690.809} C_VEL
LIN {X 0,Y 280.721,Z 367.678,A -85,B 0,C 180,E1 -17691.966,E2 -17691.966} C_VEL
LIN {X 0,Y 285.47,Z 388.984,A -85,B 0,C 180,E1 -17693.426,E2 -17693.426} C_VEL
LIN {X 0,Y 287.449,Z 403.824,A -85,B 0,C 180,E1 -17694.506,E2 -17694.506} C_VEL
LIN {X 0,Y 288.494,Z 417.85,A -85,B 0,C 180,E1 -17695.692,E2 -17695.692} C_VEL
LIN {X 0,Y 288.852,Z 432.882,A -85,B 0,C 180,E1 -17697.173,E2 -17697.173} C_VEL
LIN {X 0,Y 288.49,Z 442.758,A -85,B 0,C 180,E1 -17698.271,E2 -17698.271} C_VEL
LIN {X 0,Y 285.72,Z 455.625,A -85,B 0,C 180,E1 -17699.719,E2 -17699.719} C_VEL
LIN {X 0,Y 282.769,Z 467.897,A -85,B 0,C 180,E1 -17701.417,E2 -17701.417} C_VEL
LIN {X 0,Y 280.008,Z 478.223,A -85,B 0,C 180,E1 -17703.142,E2 -17703.142} C_VEL
LIN {X 0,Y 277.229,Z 488.798,A -85,B 0,C 180,E1 -17705.274,E2 -17705.274} C_VEL
LIN {X 0,Y 274.887,Z 497.784,A -85,B 0,C 180,E1 -17707.449,E2 -17707.449} C_VEL
LIN {X 0,Y 272.58,Z 506.634,A -85,B 0,C 180,E1 -17710.024,E2 -17710.024} C_VEL
LIN {X 0,Y 270.855,Z 514.026,A -85,B 0,C 180,E1 -17712.639,E2 -17712.639} C_VEL
LIN {X 0,Y 269.493,Z 520.903,A -85,B 0,C 180,E1 -17715.656,E2 -17715.656} C_VEL
LIN {X 0,Y 268.755,Z 526.309,A -85,B 0,C 180,E1 -17718.69,E2 -17718.69} C_VEL
LIN {X 0,Y 268.587,Z 529.44,A -85,B 0,C 180,E1 -17720.968,E2 -17720.968} C_VEL
LIN {X 0,Y 268.738,Z 532.534,A -85,B 0,C 180,E1 -17723.996,E2 -17723.996} C_VEL
LIN {X 0,Y 268.87,Z 534.382,A -85,B 0,C 180,E1 -17727.004,E2 -17727.004} C_VEL
LIN {X 0,Y 269.029,Z 534.861,A -85,B 0,C 180,E1 -17728.503,E2 -17728.503} C_VEL
LIN {X 0,Y 269.079,Z 535.025,A -85,B 0,C 180,E1 -17730,E2 -17730} C_VEL
LIN {X 0,Y 269.045,Z 534.861,A -85,B 0,C 180,E1 -17731.497,E2 -17731.497} C_VEL
LIN {X 0,Y 268.776,Z 533.599,A -85,B 0,C 180,E1 -17734.5,E2 -17734.5} C_VEL
LIN {X 0,Y 268.73,Z 532.221,A -85,B 0,C 180,E1 -17736.385,E2 -17736.385} C_VEL
LIN {X 0,Y 268.634,Z 528.474,A -85,B 0,C 180,E1 -17739.791,E2 -17739.791} C_VEL
LIN {X 0,Y 269.085,Z 523.737,A -85,B 0,C 180,E1 -17742.827,E2 -17742.827} C_VEL
LIN {X 0,Y 270.155,Z 517.362,A -85,B 0,C 180,E1 -17745.966,E2 -17745.966} C_VEL
LIN {X 0,Y 271.726,Z 509.911,A -85,B 0,C 180,E1 -17748.863,E2 -17748.863} C_VEL
LIN {X 0,Y 273.898,Z 501.7,A -85,B 0,C 180,E1 -17751.448,E2 -17751.448} C_VEL
LIN {X 0,Y 276.402,Z 491.848,A -85,B 0,C 180,E1 -17754.006,E2 -17754.006} C_VEL
LIN {X 0,Y 278.631,Z 484.049,A -85,B 0,C 180,E1 -17755.792,E2 -17755.792} C_VEL
LIN {X 0,Y 283.116,Z 473.445,A -85,B 0,C 180,E1 -17758.546,E2 -17758.546} C_VEL
LIN {X 0,Y 287.923,Z 462.746,A -85,B 0,C 180,E1 -17760.837,E2 -17760.837} C_VEL
LIN {X 0,Y 293.682,Z 449.941,A -85,B 0,C 180,E1 -17763.081,E2 -17763.081} C_VEL
LIN {X 0,Y 297.65,Z 438.689,A -85,B 0,C 180,E1 -17764.931,E2 -17764.931} C_VEL
LIN {X 0,Y 300.864,Z 426.955,A -85,B 0,C 180,E1 -17766.85,E2 -17766.85} C_VEL
LIN {X 0,Y 303.086,Z 414.638,A -85,B 0,C 180,E1 -17769.048,E2 -17769.048} C_VEL
LIN {X 0,Y 304.486,Z 403.636,A -85,B 0,C 180,E1 -17771.278,E2 -17771.278} C_VEL
LIN {X 0,Y 304.855,Z 400.573,A -85,B 0,C 180,E1 -17771.956,E2 -17771.956} C_VEL
LIN {X 0,Y 304.943,Z 398.633,A -85,B 0,C 180,E1 -17772.481,E2 -17772.481} C_VEL
LIN {X 0,Y 303.838,Z 395.554,A -85,B 0,C 180,E1 -17774.188,E2 -17774.188} C_VEL
LIN {X 0,Y 303.031,Z 393.07,A -85,B 0,C 180,E1 -17775.969,E2 -17775.969} C_VEL
LIN {X 0,Y 302.547,Z 391.147,A -85,B 0,C 180,E1 -17778.017,E2 -17778.017} C_VEL
LIN {X 0,Y 302.507,Z 390.09,A -85,B 0,C 180,E1 -17780.057,E2 -17780.057} C_VEL
LIN {X 0,Y 302.841,Z 390.099,A -85,B 0,C 180,E1 -17782.096,E2 -17782.096} C_VEL
LIN {X 0,Y 303.596,Z 391.623,A -85,B 0,C 180,E1 -17784.639,E2 -17784.639} C_VEL
LIN {X 0,Y 304.546,Z 394.367,A -85,B 0,C 180,E1 -17786.945,E2 -17786.945} C_VEL
LIN {X 0,Y 305.394,Z 397.845,A -85,B 0,C 180,E1 -17788.979,E2 -17788.979} C_VEL
LIN {X 0,Y 306.146,Z 402.613,A -85,B 0,C 180,E1 -17791.179,E2 -17791.179} C_VEL
LIN {X 0,Y 306.094,Z 403.55,A -85,B 0,C 180,E1 -17791.511,E2 -17791.511} C_VEL
LIN {X 0,Y 301.386,Z 413.142,A -85,B 0,C 180,E1 -17793.328,E2 -17793.328} C_VEL
LIN {X 0,Y 296.328,Z 422.503,A -85,B 0,C 180,E1 -17795.478,E2 -17795.478} C_VEL
LIN {X 0,Y 292.361,Z 429.202,A -85,B 0,C 180,E1 -17797.38,E2 -17797.38} C_VEL
LIN {X 0,Y 287.509,Z 436.59,A -85,B 0,C 180,E1 -17799.988,E2 -17799.988} C_VEL
LIN {X 0,Y 283.38,Z 442.341,A -85,B 0,C 180,E1 -17802.686,E2 -17802.686} C_VEL
LIN {X 0,Y 279.831,Z 446.531,A -85,B 0,C 180,E1 -17805.454,E2 -17805.454} C_VEL
LIN {X 0,Y 276.883,Z 449.273,A -85,B 0,C 180,E1 -17808.284,E2 -17808.284} C_VEL
LIN {X 0,Y 274.526,Z 450.606,A -85,B 0,C 180,E1 -17811.164,E2 -17811.164} C_VEL
LIN {X 0,Y 272.867,Z 450.518,A -85,B 0,C 180,E1 -17814.087,E2 -17814.087} C_VEL
LIN {X 0,Y 272.248,Z 449.906,A -85,B 0,C 180,E1 -17815.558,E2 -17815.558} C_VEL
LIN {X 0,Y 271.56,Z 448.956,A -85,B 0,C 180,E1 -17817.033,E2 -17817.033} C_VEL
LIN {X 0,Y 271.235,Z 447.606,A -85,B 0,C 180,E1 -17818.515,E2 -17818.515} C_VEL
LIN {X 0,Y 270.644,Z 444.9,A -85,B 0,C 180,E1 -17820.744,E2 -17820.744} C_VEL
LIN {X 0,Y 270.306,Z 441.291,A -85,B 0,C 180,E1 -17822.981,E2 -17822.981} C_VEL
LIN {X 0,Y 270.403,Z 436.715,A -85,B 0,C 180,E1 -17825.219,E2 -17825.219} C_VEL
LIN {X 0,Y 270.888,Z 429.867,A -85,B 0,C 180,E1 -17827.869,E2 -17827.869} C_VEL
LIN {X 0,Y 271.518,Z 421.653,A -85,B 0,C 180,E1 -17830.439,E2 -17830.439} C_VEL
LIN {X 0,Y 272.275,Z 412.997,A -85,B 0,C 180,E1 -17832.674,E2 -17832.674} C_VEL
LIN {X 0,Y 273.247,Z 402.578,A -85,B 0,C 180,E1 -17834.904,E2 -17834.904} C_VEL
LIN {X 0,Y 274.449,Z 391.122,A -85,B 0,C 180,E1 -17836.935,E2 -17836.935} C_VEL
LIN {X 0,Y 275.726,Z 378.473,A -85,B 0,C 180,E1 -17838.772,E2 -17838.772} C_VEL
LIN {X 0,Y 276.932,Z 365.211,A -85,B 0,C 180,E1 -17840.353,E2 -17840.353} C_VEL
LIN {X 0,Y 277.42,Z 359.65,A -85,B 0,C 180,E1 -17840.921,E2 -17840.921} C_VEL
LIN {X 0,Y 274.774,Z 347.129,A -85,B 0,C 180,E1 -17842.209,E2 -17842.209} C_VEL
LIN {X 0,Y 270.89,Z 331.034,A -85,B 0,C 180,E1 -17843.583,E2 -17843.583} C_VEL
LIN {X 0,Y 269.74,Z 326.284,A -85,B 0,C 180,E1 -17843.948,E2 -17843.948} C_VEL
LIN {X 0,Y 269.815,Z 322.362,A -85,B 0,C 180,E1 -17847.96,E2 -17847.96} C_VEL
LIN {X 0,Y 269.882,Z 318.319,A -85,B 0,C 180,E1 -17852.266,E2 -17852.266} C_VEL
LIN {X 0,Y 269.876,Z 317.944,A -85,B 0,C 180,E1 -17852.708,E2 -17852.708} C_VEL
LIN {X 0,Y 271.024,Z 321.471,A -85,B 0,C 180,E1 -17856.614,E2 -17856.614} C_VEL
LIN {X 0,Y 271.821,Z 325.053,A -85,B 0,C 180,E1 -17860.27,E2 -17860.27} C_VEL
LIN {X 0,Y 272.479,Z 329.039,A -85,B 0,C 180,E1 -17864.14,E2 -17864.14} C_VEL
LIN {X 0,Y 272.97,Z 332.257,A -85,B 0,C 180,E1 -17867.09,E2 -17867.09} C_VEL
LIN {X 0,Y 273.032,Z 336.457,A -85,B 0,C 180,E1 -17870.554,E2 -17870.554} C_VEL
LIN {X 0,Y 273.027,Z 336.778,A -85,B 0,C 180,E1 -17870.754,E2 -17870.754} C_VEL
LIN {X 0,Y 274.623,Z 340.098,A -85,B 0,C 180,E1 -17871.141,E2 -17871.141} C_VEL
LIN {X 0,Y 281.094,Z 352.644,A -85,B 0,C 180,E1 -17872.748,E2 -17872.748} C_VEL
LIN {X 0,Y 286.662,Z 365.854,A -85,B 0,C 180,E1 -17874.422,E2 -17874.422} C_VEL
LIN {X 0,Y 290.574,Z 377.56,A -85,B 0,C 180,E1 -17875.934,E2 -17875.934} C_VEL
LIN {X 0,Y 293.713,Z 389.757,A -85,B 0,C 180,E1 -17877.59,E2 -17877.59} C_VEL
LIN {X 0,Y 291.838,Z 401.923,A -85,B 0,C 180,E1 -17878.817,E2 -17878.817} C_VEL
LIN {X 0,Y 289,Z 415.74,A -85,B 0,C 180,E1 -17880.498,E2 -17880.498} C_VEL
LIN {X 0,Y 286.224,Z 427.149,A -85,B 0,C 180,E1 -17882.19,E2 -17882.19} C_VEL
LIN {X 0,Y 283.369,Z 438.586,A -85,B 0,C 180,E1 -17884.276,E2 -17884.276} C_VEL
LIN {X 0,Y 280.62,Z 448.207,A -85,B 0,C 180,E1 -17886.377,E2 -17886.377} C_VEL
LIN {X 0,Y 277.853,Z 457.594,A -85,B 0,C 180,E1 -17888.872,E2 -17888.872} C_VEL
LIN {X 0,Y 275.549,Z 465.391,A -85,B 0,C 180,E1 -17891.408,E2 -17891.408} C_VEL
LIN {X 0,Y 273.328,Z 472.64,A -85,B 0,C 180,E1 -17894.336,E2 -17894.336} C_VEL
LIN {X 0,Y 271.668,Z 478.371,A -85,B 0,C 180,E1 -17897.297,E2 -17897.297} C_VEL
LIN {X 0,Y 270.695,Z 481.752,A -85,B 0,C 180,E1 -17899.529,E2 -17899.529} C_VEL
LIN {X 0,Y 269.751,Z 485.192,A -85,B 0,C 180,E1 -17902.515,E2 -17902.515} C_VEL
LIN {X 0,Y 269.42,Z 487.434,A -85,B 0,C 180,E1 -17905.511,E2 -17905.511} C_VEL
LIN {X 0,Y 269.04,Z 488.591,A -85,B 0,C 180,E1 -17908.503,E2 -17908.503} C_VEL
LIN {X 0,Y 269.039,Z 488.602,A -85,B 0,C 180,E1 -17911.497,E2 -17911.497} C_VEL
LIN {X 0,Y 269.389,Z 487.493,A -85,B 0,C 180,E1 -17914.489,E2 -17914.489} C_VEL
LIN {X 0,Y 269.757,Z 485.296,A -85,B 0,C 180,E1 -17917.485,E2 -17917.485} C_VEL
LIN {X 0,Y 270.691,Z 481.914,A -85,B 0,C 180,E1 -17920.471,E2 -17920.471} C_VEL
LIN {X 0,Y 271.983,Z 477.276,A -85,B 0,C 180,E1 -17923.447,E2 -17923.447} C_VEL
LIN {X 0,Y 273.736,Z 471.242,A -85,B 0,C 180,E1 -17926.404,E2 -17926.404} C_VEL
LIN {X 0,Y 276.052,Z 463.631,A -85,B 0,C 180,E1 -17929.327,E2 -17929.327} C_VEL
LIN {X 0,Y 278.524,Z 455.497,A -85,B 0,C 180,E1 -17931.85,E2 -17931.85} C_VEL
LIN {X 0,Y 281.453,Z 445.665,A -85,B 0,C 180,E1 -17934.331,E2 -17934.331} C_VEL
LIN {X 0,Y 284.135,Z 435.617,A -85,B 0,C 180,E1 -17936.437,E2 -17936.437} C_VEL
LIN {X 0,Y 286.935,Z 424.67,A -85,B 0,C 180,E1 -17938.33,E2 -17938.33} C_VEL
LIN {X 0,Y 289.98,Z 411.436,A -85,B 0,C 180,E1 -17940.192,E2 -17940.192} C_VEL
LIN {X 0,Y 292.63,Z 398.18,A -85,B 0,C 180,E1 -17941.693,E2 -17941.693} C_VEL
LIN {X 0,Y 293.81,Z 389.931,A -85,B 0,C 180,E1 -17942.501,E2 -17942.501} C_VEL
LIN {X 0,Y 290.403,Z 376.742,A -85,B 0,C 180,E1 -17944.286,E2 -17944.286} C_VEL
LIN {X 0,Y 285.954,Z 363.845,A -85,B 0,C 180,E1 -17945.961,E2 -17945.961} C_VEL
LIN {X 0,Y 279.803,Z 349.921,A -85,B 0,C 180,E1 -17947.736,E2 -17947.736} C_VEL
LIN {X 0,Y 274.623,Z 340.062,A -85,B 0,C 180,E1 -17948.995,E2 -17948.995} C_VEL
LIN {X 0,Y 273.157,Z 337.152,A -85,B 0,C 180,E1 -17949.346,E2 -17949.346} C_VEL
LIN {X 0,Y 273.028,Z 336.648,A -85,B 0,C 180,E1 -17949.445,E2 -17949.445} C_VEL
LIN {X 0,Y 272.989,Z 332.445,A -85,B 0,C 180,E1 -17952.908,E2 -17952.908} C_VEL
LIN {X 0,Y 272.449,Z 328.821,A -85,B 0,C 180,E1 -17956.243,E2 -17956.243} C_VEL
LIN {X 0,Y 271.841,Z 325.225,A -85,B 0,C 180,E1 -17959.734,E2 -17959.734} C_VEL
LIN {X 0,Y 271.153,Z 321.575,A -85,B 0,C 180,E1 -17963.464,E2 -17963.464} C_VEL
LIN {X 0,Y 270.191,Z 317.452,A -85,B 0,C 180,E1 -17967.886,E2 -17967.886} C_VEL
LIN {X 0,Y 270.222,Z 317.45,A -85,B 0,C 180,E1 -17972.163,E2 -17972.163} C_VEL
LIN {X 0,Y 270.228,Z 317.446,A -85,B 0,C 180,E1 -17975.542,E2 -17975.542} C_VEL
LIN {X 0,Y 270.279,Z 317.442,A -85,B 0,C 180,E1 -17980.243,E2 -17980.243} C_VEL
LIN {X 0,Y 270.377,Z 317.425,A -85,B 0,C 180,E1 -17984.934,E2 -17984.934} C_VEL
LIN {X 0,Y 270.41,Z 317.409,A -85,B 0,C 180,E1 -17989.518,E2 -17989.518} C_VEL
LIN {X 0,Y 270.563,Z 317.392,A -85,B 0,C 180,E1 -17992.537,E2 -17992.537} C_VEL
LIN {X 0,Y 270.787,Z 317.36,A -85,B 0,C 180,E1 -17998.513,E2 -17998.513} C_VEL
LIN {X 0,Y 270.783,Z 317.371,A -85,B 0,C 180,E1 -18001.487,E2 -18001.487} C_VEL
LIN {X 0,Y 270.423,Z 317.405,A -85,B 0,C 180,E1 -18004.189,E2 -18004.189} C_VEL
LIN {X 0,Y 269.686,Z 317.497,A -85,B 0,C 180,E1 -18005.432,E2 -18005.432} C_VEL
LIN {X 0,Y 266.87,Z 317.863,A -85,B 0,C 180,E1 -18007.461,E2 -18007.461} C_VEL
LIN {X 0,Y 264.503,Z 318.154,A -85,B 0,C 180,E1 -18009.11,E2 -18009.11} C_VEL
LIN {X 0,Y 263.453,Z 318.269,A -85,B 0,C 180,E1 -18010.385,E2 -18010.385} C_VEL
LIN {X 0,Y 263.346,Z 318.28,A -85,B 0,C 180,E1 -18010.818,E2 -18010.818} C_VEL
LIN {X 0,Y 263.351,Z 318.286,A -85,B 0,C 180,E1 -18015.478,E2 -18015.478} C_VEL
LIN {X 0,Y 263.262,Z 318.304,A -85,B 0,C 180,E1 -18020.307,E2 -18020.307} C_VEL
LIN {X 0,Y 263.167,Z 318.317,A -85,B 0,C 180,E1 -18025.295,E2 -18025.295} C_VEL
LIN {X 0,Y 263.162,Z 318.331,A -85,B 0,C 180,E1 -18030.049,E2 -18030.049} C_VEL
LIN {X 0,Y 264.839,Z 325.876,A -85,B 0,C 180,E1 -18034.65,E2 -18034.65} C_VEL
LIN {X 0,Y 266.619,Z 334.038,A -85,B 0,C 180,E1 -18039.244,E2 -18039.244} C_VEL
LIN {X 0,Y 268.441,Z 342.185,A -85,B 0,C 180,E1 -18043.412,E2 -18043.412} C_VEL
LIN {X 0,Y 271.139,Z 351.713,A -85,B 0,C 180,E1 -18046.532,E2 -18046.532} C_VEL
LIN {X 0,Y 273.962,Z 361.991,A -85,B 0,C 180,E1 -18049.596,E2 -18049.596} C_VEL
LIN {X 0,Y 274.55,Z 364.134,A -85,B 0,C 180,E1 -18050.212,E2 -18050.212} C_VEL
LIN {X 0,Y 274.611,Z 367.364,A -85,B 0,C 180,E1 -18050.983,E2 -18050.983} C_VEL
LIN {X 0,Y 278.952,Z 386.8,A -85,B 0,C 180,E1 -18052.356,E2 -18052.356} C_VEL
LIN {X 0,Y 280.823,Z 398.586,A -85,B 0,C 180,E1 -18053.253,E2 -18053.253} C_VEL
LIN {X 0,Y 282.15,Z 413.335,A -85,B 0,C 180,E1 -18054.482,E2 -18054.482} C_VEL
LIN {X 0,Y 282.578,Z 427.15,A -85,B 0,C 180,E1 -18055.803,E2 -18055.803} C_VEL
LIN {X 0,Y 282.441,Z 440.364,A -85,B 0,C 180,E1 -18057.277,E2 -18057.277} C_VEL
LIN {X 0,Y 281.421,Z 447.046,A -85,B 0,C 180,E1 -18058.029,E2 -18058.029} C_VEL
LIN {X 0,Y 278.353,Z 460.219,A -85,B 0,C 180,E1 -18059.671,E2 -18059.671} C_VEL
LIN {X 0,Y 274.982,Z 472.667,A -85,B 0,C 180,E1 -18061.575,E2 -18061.575} C_VEL
LIN {X 0,Y 271.597,Z 484.887,A -85,B 0,C 180,E1 -18063.903,E2 -18063.903} C_VEL
LIN {X 0,Y 268.611,Z 495.637,A -85,B 0,C 180,E1 -18066.439,E2 -18066.439} C_VEL
LIN {X 0,Y 266.159,Z 504.882,A -85,B 0,C 180,E1 -18069.117,E2 -18069.117} C_VEL
LIN {X 0,Y 263.966,Z 513.408,A -85,B 0,C 180,E1 -18072.171,E2 -18072.171} C_VEL
LIN {X 0,Y 262.512,Z 520.285,A -85,B 0,C 180,E1 -18075.266,E2 -18075.266} C_VEL
LIN {X 0,Y 261.717,Z 525.692,A -85,B 0,C 180,E1 -18078.381,E2 -18078.381} C_VEL
LIN {X 0,Y 261.497,Z 528.823,A -85,B 0,C 180,E1 -18080.721,E2 -18080.721} C_VEL
LIN {X 0,Y 261.658,Z 531.922,A -85,B 0,C 180,E1 -18083.833,E2 -18083.833} C_VEL
LIN {X 0,Y 261.778,Z 533.772,A -85,B 0,C 180,E1 -18086.922,E2 -18086.922} C_VEL
LIN {X 0,Y 261.964,Z 534.253,A -85,B 0,C 180,E1 -18088.463,E2 -18088.463} C_VEL
LIN {X 0,Y 262.016,Z 534.418,A -85,B 0,C 180,E1 -18090,E2 -18090} C_VEL
LIN {X 0,Y 261.982,Z 534.253,A -85,B 0,C 180,E1 -18091.538,E2 -18091.538} C_VEL
LIN {X 0,Y 261.704,Z 532.989,A -85,B 0,C 180,E1 -18094.621,E2 -18094.621} C_VEL
LIN {X 0,Y 261.656,Z 531.744,A -85,B 0,C 180,E1 -18096.381,E2 -18096.381} C_VEL
LIN {X 0,Y 261.572,Z 527.857,A -85,B 0,C 180,E1 -18100.058,E2 -18100.058} C_VEL
LIN {X 0,Y 262.069,Z 523.118,A -85,B 0,C 180,E1 -18103.177,E2 -18103.177} C_VEL
LIN {X 0,Y 263.181,Z 516.969,A -85,B 0,C 180,E1 -18106.292,E2 -18106.292} C_VEL
LIN {X 0,Y 264.913,Z 509.292,A -85,B 0,C 180,E1 -18109.367,E2 -18109.367} C_VEL
LIN {X 0,Y 267.19,Z 501.081,A -85,B 0,C 180,E1 -18112.014,E2 -18112.014} C_VEL
LIN {X 0,Y 269.866,Z 491.234,A -85,B 0,C 180,E1 -18114.626,E2 -18114.626} C_VEL
LIN {X 0,Y 271.2,Z 486.66,A -85,B 0,C 180,E1 -18115.726,E2 -18115.726} C_VEL
LIN {X 0,Y 276.29,Z 475.543,A -85,B 0,C 180,E1 -18118.902,E2 -18118.902} C_VEL
LIN {X 0,Y 281.936,Z 463.928,A -85,B 0,C 180,E1 -18121.567,E2 -18121.567} C_VEL
LIN {X 0,Y 287.382,Z 452.708,A -85,B 0,C 180,E1 -18123.669,E2 -18123.669} C_VEL
LIN {X 0,Y 290.072,Z 446.679,A -85,B 0,C 180,E1 -18124.706,E2 -18124.706} C_VEL
LIN {X 0,Y 294.993,Z 432.585,A -85,B 0,C 180,E1 -18127.131,E2 -18127.131} C_VEL
LIN {X 0,Y 297.705,Z 421.538,A -85,B 0,C 180,E1 -18129.16,E2 -18129.16} C_VEL
LIN {X 0,Y 299.839,Z 410.572,A -85,B 0,C 180,E1 -18131.405,E2 -18131.405} C_VEL
LIN {X 0,Y 300.785,Z 405.072,A -85,B 0,C 180,E1 -18132.657,E2 -18132.657} C_VEL
LIN {X 0,Y 300.604,Z 402.87,A -85,B 0,C 180,E1 -18133.551,E2 -18133.551} C_VEL
LIN {X 0,Y 299.754,Z 400.167,A -85,B 0,C 180,E1 -18135.302,E2 -18135.302} C_VEL
LIN {X 0,Y 299.157,Z 398.203,A -85,B 0,C 180,E1 -18137.056,E2 -18137.056} C_VEL
LIN {X 0,Y 298.89,Z 396.83,A -85,B 0,C 180,E1 -18138.824,E2 -18138.824} C_VEL
LIN {X 0,Y 298.995,Z 396.095,A -85,B 0,C 180,E1 -18140.867,E2 -18140.867} C_VEL
LIN {X 0,Y 299.358,Z 396.484,A -85,B 0,C 180,E1 -18142.961,E2 -18142.961} C_VEL
LIN {X 0,Y 300.061,Z 398.791,A -85,B 0,C 180,E1 -18145.797,E2 -18145.797} C_VEL
LIN {X 0,Y 300.748,Z 402.413,A -85,B 0,C 180,E1 -18148.346,E2 -18148.346} C_VEL
LIN {X 0,Y 301.212,Z 406.969,A -85,B 0,C 180,E1 -18150.661,E2 -18150.661} C_VEL
LIN {X 0,Y 301.152,Z 407.417,A -85,B 0,C 180,E1 -18150.821,E2 -18150.821} C_VEL
LIN {X 0,Y 295.779,Z 417.246,A -85,B 0,C 180,E1 -18152.781,E2 -18152.781} C_VEL
LIN {X 0,Y 289.74,Z 427.156,A -85,B 0,C 180,E1 -18155.265,E2 -18155.265} C_VEL
LIN {X 0,Y 285.041,Z 434.238,A -85,B 0,C 180,E1 -18157.532,E2 -18157.532} C_VEL
LIN {X 0,Y 280.155,Z 440.759,A -85,B 0,C 180,E1 -18160.205,E2 -18160.205} C_VEL
LIN {X 0,Y 275.975,Z 445.759,A -85,B 0,C 180,E1 -18162.971,E2 -18162.971} C_VEL
LIN {X 0,Y 273.244,Z 448.523,A -85,B 0,C 180,E1 -18165.096,E2 -18165.096} C_VEL
LIN {X 0,Y 270.155,Z 450.987,A -85,B 0,C 180,E1 -18167.988,E2 -18167.988} C_VEL
LIN {X 0,Y 267.674,Z 452.062,A -85,B 0,C 180,E1 -18170.936,E2 -18170.936} C_VEL
LIN {X 0,Y 265.904,Z 451.687,A -85,B 0,C 180,E1 -18173.931,E2 -18173.931} C_VEL
LIN {X 0,Y 265.264,Z 450.964,A -85,B 0,C 180,E1 -18175.441,E2 -18175.441} C_VEL
LIN {X 0,Y 264.553,Z 449.905,A -85,B 0,C 180,E1 -18176.955,E2 -18176.955} C_VEL
LIN {X 0,Y 264.194,Z 448.451,A -85,B 0,C 180,E1 -18178.476,E2 -18178.476} C_VEL
LIN {X 0,Y 263.575,Z 445.552,A -85,B 0,C 180,E1 -18180.764,E2 -18180.764} C_VEL
LIN {X 0,Y 263.226,Z 441.75,A -85,B 0,C 180,E1 -18183.061,E2 -18183.061} C_VEL
LIN {X 0,Y 263.341,Z 436.967,A -85,B 0,C 180,E1 -18185.36,E2 -18185.36} C_VEL
LIN {X 0,Y 263.831,Z 430.069,A -85,B 0,C 180,E1 -18188.039,E2 -18188.039} C_VEL
LIN {X 0,Y 264.416,Z 422.469,A -85,B 0,C 180,E1 -18190.441,E2 -18190.441} C_VEL
LIN {X 0,Y 265.301,Z 412.54,A -85,B 0,C 180,E1 -18193.013,E2 -18193.013} C_VEL
LIN {X 0,Y 266.322,Z 401.84,A -85,B 0,C 180,E1 -18195.301,E2 -18195.301} C_VEL
LIN {X 0,Y 267.56,Z 390.031,A -85,B 0,C 180,E1 -18197.385,E2 -18197.385} C_VEL
LIN {X 0,Y 268.942,Z 377.111,A -85,B 0,C 180,E1 -18199.264,E2 -18199.264} C_VEL
LIN {X 0,Y 270.114,Z 364.605,A -85,B 0,C 180,E1 -18200.756,E2 -18200.756} C_VEL
LIN {X 0,Y 270.413,Z 360.02,A -85,B 0,C 180,E1 -18201.236,E2 -18201.236} C_VEL
LIN {X 0,Y 267.452,Z 346.716,A -85,B 0,C 180,E1 -18202.63,E2 -18202.63} C_VEL
LIN {X 0,Y 263.76,Z 331.236,A -85,B 0,C 180,E1 -18203.962,E2 -18203.962} C_VEL
LIN {X 0,Y 262.719,Z 326.9,A -85,B 0,C 180,E1 -18204.307,E2 -18204.307} C_VEL
LIN {X 0,Y 262.785,Z 322.596,A -85,B 0,C 180,E1 -18208.777,E2 -18208.777} C_VEL
LIN {X 0,Y 262.869,Z 319.82,A -85,B 0,C 180,E1 -18211.961,E2 -18211.961} C_VEL
LIN {X 0,Y 263.673,Z 321.73,A -85,B 0,C 180,E1 -18214.281,E2 -18214.281} C_VEL
LIN {X 0,Y 264.535,Z 324.799,A -85,B 0,C 180,E1 -18217.666,E2 -18217.666} C_VEL
LIN {X 0,Y 265.291,Z 328.496,A -85,B 0,C 180,E1 -18221.475,E2 -18221.475} C_VEL
LIN {X 0,Y 265.941,Z 332.712,A -85,B 0,C 180,E1 -18225.523,E2 -18225.523} C_VEL
LIN {X 0,Y 266.266,Z 336.325,A -85,B 0,C 180,E1 -18228.71,E2 -18228.71} C_VEL
LIN {X 0,Y 266.301,Z 337.473,A -85,B 0,C 180,E1 -18229.564,E2 -18229.564} C_VEL
LIN {X 0,Y 267.877,Z 340.739,A -85,B 0,C 180,E1 -18229.969,E2 -18229.969} C_VEL
LIN {X 0,Y 272.654,Z 349.632,A -85,B 0,C 180,E1 -18231.185,E2 -18231.185} C_VEL
LIN {X 0,Y 277.704,Z 360.576,A -85,B 0,C 180,E1 -18232.659,E2 -18232.659} C_VEL
LIN {X 0,Y 282.326,Z 372.744,A -85,B 0,C 180,E1 -18234.295,E2 -18234.295} C_VEL
LIN {X 0,Y 285.848,Z 384.482,A -85,B 0,C 180,E1 -18235.923,E2 -18235.923} C_VEL
LIN {X 0,Y 287.41,Z 391.194,A -85,B 0,C 180,E1 -18236.878,E2 -18236.878} C_VEL
LIN {X 0,Y 287.361,Z 393.951,A -85,B 0,C 180,E1 -18237.195,E2 -18237.195} C_VEL
LIN {X 0,Y 284.96,Z 407.024,A -85,B 0,C 180,E1 -18238.6,E2 -18238.6} C_VEL
LIN {X 0,Y 281.92,Z 420.128,A -85,B 0,C 180,E1 -18240.32,E2 -18240.32} C_VEL
LIN {X 0,Y 279.181,Z 431.016,A -85,B 0,C 180,E1 -18242.07,E2 -18242.07} C_VEL
LIN {X 0,Y 276.083,Z 442.615,A -85,B 0,C 180,E1 -18244.357,E2 -18244.357} C_VEL
LIN {X 0,Y 273.307,Z 451.695,A -85,B 0,C 180,E1 -18246.51,E2 -18246.51} C_VEL
LIN {X 0,Y 270.425,Z 460.83,A -85,B 0,C 180,E1 -18249.142,E2 -18249.142} C_VEL
LIN {X 0,Y 268.2,Z 467.952,A -85,B 0,C 180,E1 -18251.672,E2 -18251.672} C_VEL
LIN {X 0,Y 266.014,Z 474.806,A -85,B 0,C 180,E1 -18254.68,E2 -18254.68} C_VEL
LIN {X 0,Y 264.403,Z 480.176,A -85,B 0,C 180,E1 -18257.722,E2 -18257.722} C_VEL
LIN {X 0,Y 263.211,Z 484.23,A -85,B 0,C 180,E1 -18260.781,E2 -18260.781} C_VEL
LIN {X 0,Y 262.403,Z 487.073,A -85,B 0,C 180,E1 -18263.85,E2 -18263.85} C_VEL
LIN {X 0,Y 262.359,Z 488.043,A -85,B 0,C 180,E1 -18265.39,E2 -18265.39} C_VEL
LIN {X 0,Y 261.987,Z 489.198,A -85,B 0,C 180,E1 -18268.462,E2 -18268.462} C_VEL
LIN {X 0,Y 261.986,Z 489.209,A -85,B 0,C 180,E1 -18271.537,E2 -18271.537} C_VEL
LIN {X 0,Y 262.331,Z 488.101,A -85,B 0,C 180,E1 -18274.61,E2 -18274.61} C_VEL
LIN {X 0,Y 262.755,Z 485.903,A -85,B 0,C 180,E1 -18277.685,E2 -18277.685} C_VEL
LIN {X 0,Y 263.729,Z 482.522,A -85,B 0,C 180,E1 -18280.751,E2 -18280.751} C_VEL
LIN {X 0,Y 265.089,Z 477.883,A -85,B 0,C 180,E1 -18283.804,E2 -18283.804} C_VEL
LIN {X 0,Y 266.939,Z 471.849,A -85,B 0,C 180,E1 -18286.834,E2 -18286.834} C_VEL
LIN {X 0,Y 269.367,Z 464.237,A -85,B 0,C 180,E1 -18289.827,E2 -18289.827} C_VEL
LIN {X 0,Y 271.952,Z 456.101,A -85,B 0,C 180,E1 -18292.407,E2 -18292.407} C_VEL
LIN {X 0,Y 275.013,Z 446.266,A -85,B 0,C 180,E1 -18294.939,E2 -18294.939} C_VEL
LIN {X 0,Y 277.789,Z 436.218,A -85,B 0,C 180,E1 -18297.09,E2 -18297.09} C_VEL
LIN {X 0,Y 280.728,Z 425.265,A -85,B 0,C 180,E1 -18299.016,E2 -18299.016} C_VEL
LIN {X 0,Y 283.895,Z 412.025,A -85,B 0,C 180,E1 -18300.909,E2 -18300.909} C_VEL
LIN {X 0,Y 286.646,Z 398.762,A -85,B 0,C 180,E1 -18302.434,E2 -18302.434} C_VEL
LIN {X 0,Y 287.674,Z 391.909,A -85,B 0,C 180,E1 -18303.13,E2 -18303.13} C_VEL
LIN {X 0,Y 284.286,Z 378.547,A -85,B 0,C 180,E1 -18305.025,E2 -18305.025} C_VEL
LIN {X 0,Y 279.634,Z 365.189,A -85,B 0,C 180,E1 -18306.854,E2 -18306.854} C_VEL
LIN {X 0,Y 274.935,Z 354.229,A -85,B 0,C 180,E1 -18308.316,E2 -18308.316} C_VEL
LIN {X 0,Y 268.279,Z 341.312,A -85,B 0,C 180,E1 -18310.075,E2 -18310.075} C_VEL
LIN {X 0,Y 266.547,Z 338.246,A -85,B 0,C 180,E1 -18310.502,E2 -18310.502} C_VEL
LIN {X 0,Y 266.255,Z 337.319,A -85,B 0,C 180,E1 -18310.617,E2 -18310.617} C_VEL
LIN {X 0,Y 266.151,Z 334.097,A -85,B 0,C 180,E1 -18313.358,E2 -18313.358} C_VEL
LIN {X 0,Y 265.426,Z 329.389,A -85,B 0,C 180,E1 -18317.85,E2 -18317.85} C_VEL
LIN {X 0,Y 264.981,Z 326.774,A -85,B 0,C 180,E1 -18320.465,E2 -18320.465} C_VEL
LIN {X 0,Y 264.28,Z 323.28,A -85,B 0,C 180,E1 -18324.194,E2 -18324.194} C_VEL
LIN {X 0,Y 263.559,Z 319.972,A -85,B 0,C 180,E1 -18327.77,E2 -18327.77} C_VEL
LIN {X 0,Y 263.139,Z 318.319,A -85,B 0,C 180,E1 -18329.727,E2 -18329.727} C_VEL
LIN {X 0,Y 263.14,Z 318.32,A -85,B 0,C 180,E1 -18332.997,E2 -18332.997} C_VEL
LIN {X 0,Y 263.147,Z 318.33,A -85,B 0,C 180,E1 -18336.383,E2 -18336.383} C_VEL
LIN {X 0,Y 263.244,Z 318.309,A -85,B 0,C 180,E1 -18339.692,E2 -18339.692} C_VEL
LIN {X 0,Y 263.323,Z 318.296,A -85,B 0,C 180,E1 -18344.52,E2 -18344.52} C_VEL
LIN {X 0,Y 263.349,Z 318.285,A -85,B 0,C 180,E1 -18349.233,E2 -18349.233} C_VEL
LIN {X 0,Y 263.526,Z 318.271,A -85,B 0,C 180,E1 -18352.337,E2 -18352.337} C_VEL
LIN {X 0,Y 263.751,Z 318.236,A -85,B 0,C 180,E1 -18358.473,E2 -18358.473} C_VEL
LIN {X 0,Y 263.747,Z 318.247,A -85,B 0,C 180,E1 -18361.527,E2 -18361.527} C_VEL
LIN {X 0,Y 263.536,Z 318.281,A -85,B 0,C 180,E1 -18367.663,E2 -18367.663} C_VEL
LIN {X 0,Y 263.346,Z 318.28,A -85,B 0,C 180,E1 -18370.818,E2 -18370.818} C_VEL
LIN {X 0,Y 262.628,Z 318.377,A -85,B 0,C 180,E1 -18372.093,E2 -18372.093} C_VEL
LIN {X 0,Y 259.788,Z 318.749,A -85,B 0,C 180,E1 -18374.173,E2 -18374.173} C_VEL
LIN {X 0,Y 257.384,Z 319.038,A -85,B 0,C 180,E1 -18375.864,E2 -18375.864} C_VEL
LIN {X 0,Y 256.316,Z 319.163,A -85,B 0,C 180,E1 -18377.174,E2 -18377.174} C_VEL
LIN {X 0,Y 256.206,Z 319.177,A -85,B 0,C 180,E1 -18377.618,E2 -18377.618} C_VEL
LIN {X 0,Y 256.152,Z 319.182,A -85,B 0,C 180,E1 -18381.117,E2 -18381.117} C_VEL
LIN {X 0,Y 256.132,Z 319.195,A -85,B 0,C 180,E1 -18385.112,E2 -18385.112} C_VEL
LIN {X 0,Y 256.128,Z 319.386,A -85,B 0,C 180,E1 -18389.45,E2 -18389.45} C_VEL
LIN {X 0,Y 257.725,Z 326.568,A -85,B 0,C 180,E1 -18393.988,E2 -18393.988} C_VEL
LIN {X 0,Y 259.417,Z 334.408,A -85,B 0,C 180,E1 -18398.543,E2 -18398.543} C_VEL
LIN {X 0,Y 259.841,Z 336.251,A -85,B 0,C 180,E1 -18399.465,E2 -18399.465} C_VEL
LIN {X 0,Y 262.764,Z 347.053,A -85,B 0,C 180,E1 -18403.533,E2 -18403.533} C_VEL
LIN {X 0,Y 265.172,Z 355.702,A -85,B 0,C 180,E1 -18406.442,E2 -18406.442} C_VEL
LIN {X 0,Y 268.052,Z 366.44,A -85,B 0,C 180,E1 -18409.784,E2 -18409.784} C_VEL
LIN {X 0,Y 269.463,Z 370.963,A -85,B 0,C 180,E1 -18410.226,E2 -18410.226} C_VEL
LIN {X 0,Y 273.301,Z 388.584,A -85,B 0,C 180,E1 -18411.547,E2 -18411.547} C_VEL
LIN {X 0,Y 275.094,Z 401.121,A -85,B 0,C 180,E1 -18412.553,E2 -18412.553} C_VEL
LIN {X 0,Y 276.161,Z 415.205,A -85,B 0,C 180,E1 -18413.803,E2 -18413.803} C_VEL
LIN {X 0,Y 276.355,Z 430.152,A -85,B 0,C 180,E1 -18415.32,E2 -18415.32} C_VEL
LIN {X 0,Y 276.015,Z 442.666,A -85,B 0,C 180,E1 -18416.809,E2 -18416.809} C_VEL
LIN {X 0,Y 273.718,Z 453.623,A -85,B 0,C 180,E1 -18418.106,E2 -18418.106} C_VEL
LIN {X 0,Y 270.263,Z 466.69,A -85,B 0,C 180,E1 -18419.962,E2 -18419.962} C_VEL
LIN {X 0,Y 266.718,Z 478.913,A -85,B 0,C 180,E1 -18422.115,E2 -18422.115} C_VEL
LIN {X 0,Y 263.752,Z 489.216,A -85,B 0,C 180,E1 -18424.342,E2 -18424.342} C_VEL
LIN {X 0,Y 260.842,Z 499.294,A -85,B 0,C 180,E1 -18427.003,E2 -18427.003} C_VEL
LIN {X 0,Y 258.424,Z 507.68,A -85,B 0,C 180,E1 -18429.712,E2 -18429.712} C_VEL
LIN {X 0,Y 256.667,Z 514.652,A -85,B 0,C 180,E1 -18432.471,E2 -18432.471} C_VEL
LIN {X 0,Y 255.264,Z 521.14,A -85,B 0,C 180,E1 -18435.654,E2 -18435.654} C_VEL
LIN {X 0,Y 254.557,Z 526.187,A -85,B 0,C 180,E1 -18438.857,E2 -18438.857} C_VEL
LIN {X 0,Y 254.413,Z 529.911,A -85,B 0,C 180,E1 -18442.061,E2 -18442.061} C_VEL
LIN {X 0,Y 254.564,Z 531.309,A -85,B 0,C 180,E1 -18443.66,E2 -18443.66} C_VEL
LIN {X 0,Y 254.687,Z 533.161,A -85,B 0,C 180,E1 -18446.837,E2 -18446.837} C_VEL
LIN {X 0,Y 254.899,Z 533.645,A -85,B 0,C 180,E1 -18448.42,E2 -18448.42} C_VEL
LIN {X 0,Y 254.956,Z 533.81,A -85,B 0,C 180,E1 -18450,E2 -18450} C_VEL
LIN {X 0,Y 254.918,Z 533.645,A -85,B 0,C 180,E1 -18451.58,E2 -18451.58} C_VEL
LIN {X 0,Y 254.633,Z 532.378,A -85,B 0,C 180,E1 -18454.75,E2 -18454.75} C_VEL
LIN {X 0,Y 254.584,Z 531.265,A -85,B 0,C 180,E1 -18456.38,E2 -18456.38} C_VEL
LIN {X 0,Y 254.467,Z 528.181,A -85,B 0,C 180,E1 -18459.539,E2 -18459.539} C_VEL
LIN {X 0,Y 254.865,Z 523.788,A -85,B 0,C 180,E1 -18462.745,E2 -18462.745} C_VEL
LIN {X 0,Y 255.965,Z 517.784,A -85,B 0,C 180,E1 -18466.057,E2 -18466.057} C_VEL
LIN {X 0,Y 257.573,Z 510.737,A -85,B 0,C 180,E1 -18469.113,E2 -18469.113} C_VEL
LIN {X 0,Y 259.816,Z 502.973,A -85,B 0,C 180,E1 -18471.836,E2 -18471.836} C_VEL
LIN {X 0,Y 262.539,Z 493.313,A -85,B 0,C 180,E1 -18474.604,E2 -18474.604} C_VEL
LIN {X 0,Y 264.012,Z 488.471,A -85,B 0,C 180,E1 -18475.843,E2 -18475.843} C_VEL
LIN {X 0,Y 268.836,Z 478.732,A -85,B 0,C 180,E1 -18478.923,E2 -18478.923} C_VEL
LIN {X 0,Y 273.731,Z 469.468,A -85,B 0,C 180,E1 -18481.327,E2 -18481.327} C_VEL
LIN {X 0,Y 280.188,Z 457.228,A -85,B 0,C 180,E1 -18483.935,E2 -18483.935} C_VEL
LIN {X 0,Y 284.343,Z 449.039,A -85,B 0,C 180,E1 -18485.423,E2 -18485.423} C_VEL
LIN {X 0,Y 289.468,Z 436.203,A -85,B 0,C 180,E1 -18487.762,E2 -18487.762} C_VEL
LIN {X 0,Y 292.288,Z 427.146,A -85,B 0,C 180,E1 -18489.482,E2 -18489.482} C_VEL
LIN {X 0,Y 294.765,Z 417.591,A -85,B 0,C 180,E1 -18491.486,E2 -18491.486} C_VEL
LIN {X 0,Y 296.369,Z 410.826,A -85,B 0,C 180,E1 -18493.042,E2 -18493.042} C_VEL
LIN {X 0,Y 296.623,Z 409.533,A -85,B 0,C 180,E1 -18493.402,E2 -18493.402} C_VEL
LIN {X 0,Y 296.513,Z 408.307,A -85,B 0,C 180,E1 -18493.962,E2 -18493.962} C_VEL
LIN {X 0,Y 295.574,Z 404.966,A -85,B 0,C 180,E1 -18496.406,E2 -18496.406} C_VEL
LIN {X 0,Y 295.179,Z 403.375,A -85,B 0,C 180,E1 -18498.19,E2 -18498.19} C_VEL
LIN {X 0,Y 295.095,Z 402.379,A -85,B 0,C 180,E1 -18499.982,E2 -18499.982} C_VEL
LIN {X 0,Y 295.228,Z 402.12,A -85,B 0,C 180,E1 -18501.775,E2 -18501.775} C_VEL
LIN {X 0,Y 295.493,Z 402.996,A -85,B 0,C 180,E1 -18503.965,E2 -18503.965} C_VEL
LIN {X 0,Y 295.911,Z 405.06,A -85,B 0,C 180,E1 -18506.23,E2 -18506.23} C_VEL
LIN {X 0,Y 296.173,Z 408.636,A -85,B 0,C 180,E1 -18508.679,E2 -18508.679} C_VEL
LIN {X 0,Y 296.15,Z 411.387,A -85,B 0,C 180,E1 -18510.109,E2 -18510.109} C_VEL
LIN {X 0,Y 290.187,Z 421.259,A -85,B 0,C 180,E1 -18512.211,E2 -18512.211} C_VEL
LIN {X 0,Y 284.662,Z 429.56,A -85,B 0,C 180,E1 -18514.402,E2 -18514.402} C_VEL
LIN {X 0,Y 278.991,Z 437.24,A -85,B 0,C 180,E1 -18517.017,E2 -18517.017} C_VEL
LIN {X 0,Y 273.906,Z 443.363,A -85,B 0,C 180,E1 -18519.734,E2 -18519.734} C_VEL
LIN {X 0,Y 270.546,Z 446.945,A -85,B 0,C 180,E1 -18521.837,E2 -18521.837} C_VEL
LIN {X 0,Y 266.68,Z 450.52,A -85,B 0,C 180,E1 -18524.72,E2 -18524.72} C_VEL
LIN {X 0,Y 263.413,Z 452.673,A -85,B 0,C 180,E1 -18527.676,E2 -18527.676} C_VEL
LIN {X 0,Y 260.815,Z 453.457,A -85,B 0,C 180,E1 -18530.696,E2 -18530.696} C_VEL
LIN {X 0,Y 258.942,Z 452.843,A -85,B 0,C 180,E1 -18533.768,E2 -18533.768} C_VEL
LIN {X 0,Y 258.279,Z 452,A -85,B 0,C 180,E1 -18535.318,E2 -18535.318} C_VEL
LIN {X 0,Y 257.545,Z 450.824,A -85,B 0,C 180,E1 -18536.872,E2 -18536.872} C_VEL
LIN {X 0,Y 257.153,Z 449.225,A -85,B 0,C 180,E1 -18538.434,E2 -18538.434} C_VEL
LIN {X 0,Y 256.508,Z 446.171,A -85,B 0,C 180,E1 -18540.785,E2 -18540.785} C_VEL
LIN {X 0,Y 256.149,Z 442.182,A -85,B 0,C 180,E1 -18543.146,E2 -18543.146} C_VEL
LIN {X 0,Y 256.285,Z 437.193,A -85,B 0,C 180,E1 -18545.508,E2 -18545.508} C_VEL
LIN {X 0,Y 256.737,Z 430.802,A -85,B 0,C 180,E1 -18547.994,E2 -18547.994} C_VEL
LIN {X 0,Y 257.343,Z 422.927,A -85,B 0,C 180,E1 -18550.529,E2 -18550.529} C_VEL
LIN {X 0,Y 258.184,Z 413.702,A -85,B 0,C 180,E1 -18552.978,E2 -18552.978} C_VEL
LIN {X 0,Y 259.212,Z 403.005,A -85,B 0,C 180,E1 -18555.329,E2 -18555.329} C_VEL
LIN {X 0,Y 260.491,Z 391.234,A -85,B 0,C 180,E1 -18557.467,E2 -18557.467} C_VEL
LIN {X 0,Y 261.871,Z 378.343,A -85,B 0,C 180,E1 -18559.397,E2 -18559.397} C_VEL
LIN {X 0,Y 263.22,Z 364.119,A -85,B 0,C 180,E1 -18561.127,E2 -18561.127} C_VEL
LIN {X 0,Y 263.306,Z 360.45,A -85,B 0,C 180,E1 -18561.531,E2 -18561.531} C_VEL
LIN {X 0,Y 259.866,Z 345.257,A -85,B 0,C 180,E1 -18563.143,E2 -18563.143} C_VEL
LIN {X 0,Y 256.321,Z 330.322,A -85,B 0,C 180,E1 -18564.428,E2 -18564.428} C_VEL
LIN {X 0,Y 255.688,Z 327.541,A -85,B 0,C 180,E1 -18564.644,E2 -18564.644} C_VEL
LIN {X 0,Y 255.754,Z 323.922,A -85,B 0,C 180,E1 -18568.436,E2 -18568.436} C_VEL
LIN {X 0,Y 255.812,Z 321.563,A -85,B 0,C 180,E1 -18571.006,E2 -18571.006} C_VEL
LIN {X 0,Y 256.644,Z 323.275,A -85,B 0,C 180,E1 -18573.209,E2 -18573.209} C_VEL
LIN {X 0,Y 257.667,Z 326.432,A -85,B 0,C 180,E1 -18576.875,E2 -18576.875} C_VEL
LIN {X 0,Y 258.423,Z 330.051,A -85,B 0,C 180,E1 -18580.746,E2 -18580.746} C_VEL
LIN {X 0,Y 259.085,Z 334.232,A -85,B 0,C 180,E1 -18584.853,E2 -18584.853} C_VEL
LIN {X 0,Y 259.485,Z 338.06,A -85,B 0,C 180,E1 -18588.266,E2 -18588.266} C_VEL
LIN {X 0,Y 261.211,Z 341.489,A -85,B 0,C 180,E1 -18588.734,E2 -18588.734} C_VEL
LIN {X 0,Y 267.538,Z 353.151,A -85,B 0,C 180,E1 -18590.457,E2 -18590.457} C_VEL
LIN {X 0,Y 272.976,Z 365.49,A -85,B 0,C 180,E1 -18592.2,E2 -18592.2} C_VEL
LIN {X 0,Y 277.057,Z 377.008,A -85,B 0,C 180,E1 -18593.848,E2 -18593.848} C_VEL
LIN {X 0,Y 280.592,Z 389.968,A -85,B 0,C 180,E1 -18595.746,E2 -18595.746} C_VEL
LIN {X 0,Y 281.444,Z 394.383,A -85,B 0,C 180,E1 -18596.394,E2 -18596.394} C_VEL
LIN {X 0,Y 278.951,Z 407.622,A -85,B 0,C 180,E1 -18597.843,E2 -18597.843} C_VEL
LIN {X 0,Y 275.796,Z 420.729,A -85,B 0,C 180,E1 -18599.592,E2 -18599.592} C_VEL
LIN {X 0,Y 272.906,Z 431.782,A -85,B 0,C 180,E1 -18601.403,E2 -18601.403} C_VEL
LIN {X 0,Y 269.719,Z 443.22,A -85,B 0,C 180,E1 -18603.706,E2 -18603.706} C_VEL
LIN {X 0,Y 266.827,Z 452.302,A -85,B 0,C 180,E1 -18605.904,E2 -18605.904} C_VEL
LIN {X 0,Y 263.765,Z 461.577,A -85,B 0,C 180,E1 -18608.637,E2 -18608.637} C_VEL
LIN {X 0,Y 261.491,Z 468.56,A -85,B 0,C 180,E1 -18611.184,E2 -18611.184} C_VEL
LIN {X 0,Y 259.193,Z 475.415,A -85,B 0,C 180,E1 -18614.267,E2 -18614.267} C_VEL
LIN {X 0,Y 257.471,Z 480.786,A -85,B 0,C 180,E1 -18617.386,E2 -18617.386} C_VEL
LIN {X 0,Y 256.223,Z 484.84,A -85,B 0,C 180,E1 -18620.527,E2 -18620.527} C_VEL
LIN {X 0,Y 255.365,Z 487.683,A -85,B 0,C 180,E1 -18623.679,E2 -18623.679} C_VEL
LIN {X 0,Y 255.13,Z 489.361,A -85,B 0,C 180,E1 -18626.841,E2 -18626.841} C_VEL
LIN {X 0,Y 254.872,Z 489.958,A -85,B 0,C 180,E1 -18630,E2 -18630} C_VEL
LIN {X 0,Y 255.123,Z 489.394,A -85,B 0,C 180,E1 -18633.158,E2 -18633.158} C_VEL
LIN {X 0,Y 255.355,Z 487.761,A -85,B 0,C 180,E1 -18636.32,E2 -18636.32} C_VEL
LIN {X 0,Y 256.222,Z 484.969,A -85,B 0,C 180,E1 -18639.472,E2 -18639.472} C_VEL
LIN {X 0,Y 257.426,Z 480.976,A -85,B 0,C 180,E1 -18642.615,E2 -18642.615} C_VEL
LIN {X 0,Y 259.163,Z 475.653,A -85,B 0,C 180,E1 -18645.734,E2 -18645.734} C_VEL
LIN {X 0,Y 261.445,Z 468.852,A -85,B 0,C 180,E1 -18648.819,E2 -18648.819} C_VEL
LIN {X 0,Y 263.754,Z 461.682,A -85,B 0,C 180,E1 -18651.451,E2 -18651.451} C_VEL
LIN {X 0,Y 266.732,Z 452.741,A -85,B 0,C 180,E1 -18654.104,E2 -18654.104} C_VEL
LIN {X 0,Y 270.113,Z 442.05,A -85,B 0,C 180,E1 -18656.668,E2 -18656.668} C_VEL
LIN {X 0,Y 272.848,Z 431.948,A -85,B 0,C 180,E1 -18658.696,E2 -18658.696} C_VEL
LIN {X 0,Y 276.052,Z 420.165,A -85,B 0,C 180,E1 -18660.609,E2 -18660.609} C_VEL
LIN {X 0,Y 279.117,Z 407.065,A -85,B 0,C 180,E1 -18662.348,E2 -18662.348} C_VEL
LIN {X 0,Y 281.554,Z 394.515,A -85,B 0,C 180,E1 -18663.7,E2 -18663.7} C_VEL
LIN {X 0,Y 278.865,Z 382.839,A -85,B 0,C 180,E1 -18665.426,E2 -18665.426} C_VEL
LIN {X 0,Y 274.811,Z 370.34,A -85,B 0,C 180,E1 -18667.238,E2 -18667.238} C_VEL
LIN {X 0,Y 269.968,Z 358.368,A -85,B 0,C 180,E1 -18668.947,E2 -18668.947} C_VEL
LIN {X 0,Y 263.675,Z 345.755,A -85,B 0,C 180,E1 -18670.759,E2 -18670.759} C_VEL
LIN {X 0,Y 261.089,Z 341.385,A -85,B 0,C 180,E1 -18671.437,E2 -18671.437} C_VEL
LIN {X 0,Y 259.452,Z 337.986,A -85,B 0,C 180,E1 -18671.935,E2 -18671.935} C_VEL
LIN {X 0,Y 259.119,Z 334.449,A -85,B 0,C 180,E1 -18675.155,E2 -18675.155} C_VEL
LIN {X 0,Y 258.46,Z 330.278,A -85,B 0,C 180,E1 -18679.262,E2 -18679.262} C_VEL
LIN {X 0,Y 257.78,Z 326.578,A -85,B 0,C 180,E1 -18683.144,E2 -18683.144} C_VEL
LIN {X 0,Y 257.072,Z 323.284,A -85,B 0,C 180,E1 -18686.854,E2 -18686.854} C_VEL
LIN {X 0,Y 256.117,Z 319.209,A -85,B 0,C 180,E1 -18691.797,E2 -18691.797} C_VEL
LIN {X 0,Y 256.134,Z 319.203,A -85,B 0,C 180,E1 -18695.696,E2 -18695.696} C_VEL
LIN {X 0,Y 256.148,Z 319.186,A -85,B 0,C 180,E1 -18699.103,E2 -18699.103} C_VEL
LIN {X 0,Y 256.259,Z 319.171,A -85,B 0,C 180,E1 -18704.082,E2 -18704.082} C_VEL
LIN {X 0,Y 256.29,Z 319.162,A -85,B 0,C 180,E1 -18708.933,E2 -18708.933} C_VEL
LIN {X 0,Y 256.49,Z 319.15,A -85,B 0,C 180,E1 -18712.125,E2 -18712.125} C_VEL
LIN {X 0,Y 256.492,Z 319.162,A -85,B 0,C 180,E1 -18716.858,E2 -18716.858} C_VEL
LIN {X 0,Y 256.758,Z 319.1,A -85,B 0,C 180,E1 -18720,E2 -18720} C_VEL
LIN {X 0,Y 256.482,Z 319.157,A -85,B 0,C 180,E1 -18723.141,E2 -18723.141} C_VEL
LIN {X 0,Y 256.497,Z 319.16,A -85,B 0,C 180,E1 -18727.874,E2 -18727.874} C_VEL
LIN {X 0,Y 256.285,Z 319.173,A -85,B 0,C 180,E1 -18732.672,E2 -18732.672} C_VEL
LIN {X 0,Y 256.283,Z 319.161,A -85,B 0,C 180,E1 -18736.302,E2 -18736.302} C_VEL
LIN {X 0,Y 256.206,Z 319.177,A -85,B 0,C 180,E1 -18737.618,E2 -18737.618} C_VEL
LIN {X 0,Y 255.46,Z 319.29,A -85,B 0,C 180,E1 -18738.929,E2 -18738.929} C_VEL
LIN {X 0,Y 252.529,Z 319.64,A -85,B 0,C 180,E1 -18741.064,E2 -18741.064} C_VEL
LIN {X 0,Y 250.112,Z 319.939,A -85,B 0,C 180,E1 -18742.803,E2 -18742.803} C_VEL
LIN {X 0,Y 249.125,Z 320.08,A -85,B 0,C 180,E1 -18744.152,E2 -18744.152} C_VEL
LIN {X 0,Y 249.068,Z 320.072,A -85,B 0,C 180,E1 -18744.609,E2 -18744.609} C_VEL
LIN {X 0,Y 249.078,Z 320.228,A -85,B 0,C 180,E1 -18748.664,E2 -18748.664} C_VEL
LIN {X 0,Y 250.719,Z 327.594,A -85,B 0,C 180,E1 -18753.193,E2 -18753.193} C_VEL
LIN {X 0,Y 253.566,Z 338.406,A -85,B 0,C 180,E1 -18758.433,E2 -18758.433} C_VEL
LIN {X 0,Y 256.75,Z 350.442,A -85,B 0,C 180,E1 -18763.182,E2 -18763.182} C_VEL
LIN {X 0,Y 258.875,Z 358.424,A -85,B 0,C 180,E1 -18766.007,E2 -18766.007} C_VEL
LIN {X 0,Y 260.801,Z 365.967,A -85,B 0,C 180,E1 -18768.472,E2 -18768.472} C_VEL
LIN {X 0,Y 263.829,Z 372.147,A -85,B 0,C 180,E1 -18769.258,E2 -18769.258} C_VEL
LIN {X 0,Y 267.556,Z 389.59,A -85,B 0,C 180,E1 -18770.647,E2 -18770.647} C_VEL
LIN {X 0,Y 269.361,Z 403.453,A -85,B 0,C 180,E1 -18771.819,E2 -18771.819} C_VEL
LIN {X 0,Y 270.259,Z 418.73,A -85,B 0,C 180,E1 -18773.266,E2 -18773.266} C_VEL
LIN {X 0,Y 270.178,Z 433.32,A -85,B 0,C 180,E1 -18774.854,E2 -18774.854} C_VEL
LIN {X 0,Y 269.512,Z 445.257,A -85,B 0,C 180,E1 -18776.349,E2 -18776.349} C_VEL
LIN {X 0,Y 266.097,Z 459.02,A -85,B 0,C 180,E1 -18778.114,E2 -18778.114} C_VEL
LIN {X 0,Y 262.485,Z 471.46,A -85,B 0,C 180,E1 -18780.087,E2 -18780.087} C_VEL
LIN {X 0,Y 258.754,Z 483.666,A -85,B 0,C 180,E1 -18782.501,E2 -18782.501} C_VEL
LIN {X 0,Y 255.894,Z 493.091,A -85,B 0,C 180,E1 -18784.793,E2 -18784.793} C_VEL
LIN {X 0,Y 253.088,Z 502.446,A -85,B 0,C 180,E1 -18787.554,E2 -18787.554} C_VEL
LIN {X 0,Y 250.784,Z 510.194,A -85,B 0,C 180,E1 -18790.349,E2 -18790.349} C_VEL
LIN {X 0,Y 248.893,Z 517.771,A -85,B 0,C 180,E1 -18793.752,E2 -18793.752} C_VEL
LIN {X 0,Y 247.831,Z 523.219,A -85,B 0,C 180,E1 -18796.888,E2 -18796.888} C_VEL
LIN {X 0,Y 247.354,Z 527.592,A -85,B 0,C 180,E1 -18800.185,E2 -18800.185} C_VEL
LIN {X 0,Y 247.481,Z 530.846,A -85,B 0,C 180,E1 -18803.684,E2 -18803.684} C_VEL
LIN {X 0,Y 247.598,Z 532.551,A -85,B 0,C 180,E1 -18806.746,E2 -18806.746} C_VEL
LIN {X 0,Y 247.834,Z 533.037,A -85,B 0,C 180,E1 -18808.375,E2 -18808.375} C_VEL
LIN {X 0,Y 247.897,Z 533.203,A -85,B 0,C 180,E1 -18810,E2 -18810} C_VEL
LIN {X 0,Y 247.853,Z 533.037,A -85,B 0,C 180,E1 -18811.625,E2 -18811.625} C_VEL
LIN {X 0,Y 247.563,Z 531.768,A -85,B 0,C 180,E1 -18814.886,E2 -18814.886} C_VEL
LIN {X 0,Y 247.494,Z 530.681,A -85,B 0,C 180,E1 -18816.522,E2 -18816.522} C_VEL
LIN {X 0,Y 247.389,Z 527.563,A -85,B 0,C 180,E1 -18819.815,E2 -18819.815} C_VEL
LIN {X 0,Y 247.854,Z 523.169,A -85,B 0,C 180,E1 -18823.112,E2 -18823.112} C_VEL
LIN {X 0,Y 248.993,Z 517.408,A -85,B 0,C 180,E1 -18826.395,E2 -18826.395} C_VEL
LIN {X 0,Y 250.774,Z 510.118,A -85,B 0,C 180,E1 -18829.652,E2 -18829.652} C_VEL
LIN {X 0,Y 253.143,Z 502.355,A -85,B 0,C 180,E1 -18832.442,E2 -18832.442} C_VEL
LIN {X 0,Y 255.883,Z 493.125,A -85,B 0,C 180,E1 -18835.165,E2 -18835.165} C_VEL
LIN {X 0,Y 256.869,Z 490.17,A -85,B 0,C 180,E1 -18835.962,E2 -18835.962} C_VEL
LIN {X 0,Y 262.04,Z 480.528,A -85,B 0,C 180,E1 -18839.306,E2 -18839.306} C_VEL
LIN {X 0,Y 267.76,Z 470.488,A -85,B 0,C 180,E1 -18842.108,E2 -18842.108} C_VEL
LIN {X 0,Y 274.467,Z 458.82,A -85,B 0,C 180,E1 -18844.743,E2 -18844.743} C_VEL
LIN {X 0,Y 278.703,Z 451.208,A -85,B 0,C 180,E1 -18846.202,E2 -18846.202} C_VEL
LIN {X 0,Y 284.352,Z 438.672,A -85,B 0,C 180,E1 -18848.615,E2 -18848.615} C_VEL
LIN {X 0,Y 287.442,Z 430.357,A -85,B 0,C 180,E1 -18850.282,E2 -18850.282} C_VEL
LIN {X 0,Y 290.706,Z 419.91,A -85,B 0,C 180,E1 -18852.604,E2 -18852.604} C_VEL
LIN {X 0,Y 292.192,Z 414.956,A -85,B 0,C 180,E1 -18853.815,E2 -18853.815} C_VEL
LIN {X 0,Y 292.276,Z 413.922,A -85,B 0,C 180,E1 -18854.213,E2 -18854.213} C_VEL
LIN {X 0,Y 291.608,Z 411.047,A -85,B 0,C 180,E1 -18856.305,E2 -18856.305} C_VEL
LIN {X 0,Y 291.181,Z 409.121,A -85,B 0,C 180,E1 -18858.437,E2 -18858.437} C_VEL
LIN {X 0,Y 291.087,Z 408.04,A -85,B 0,C 180,E1 -18861.116,E2 -18861.116} C_VEL
LIN {X 0,Y 291.208,Z 408.269,A -85,B 0,C 180,E1 -18862.89,E2 -18862.89} C_VEL
LIN {X 0,Y 291.359,Z 409.571,A -85,B 0,C 180,E1 -18865.098,E2 -18865.098} C_VEL
LIN {X 0,Y 291.43,Z 412.431,A -85,B 0,C 180,E1 -18867.571,E2 -18867.571} C_VEL
LIN {X 0,Y 291.36,Z 414.146,A -85,B 0,C 180,E1 -18868.7,E2 -18868.7} C_VEL
LIN {X 0,Y 290.794,Z 416.069,A -85,B 0,C 180,E1 -18869.5,E2 -18869.5} C_VEL
LIN {X 0,Y 284.611,Z 425.248,A -85,B 0,C 180,E1 -18871.618,E2 -18871.618} C_VEL
LIN {X 0,Y 278.882,Z 432.974,A -85,B 0,C 180,E1 -18873.832,E2 -18873.832} C_VEL
LIN {X 0,Y 272.965,Z 440.246,A -85,B 0,C 180,E1 -18876.48,E2 -18876.48} C_VEL
LIN {X 0,Y 267.683,Z 445.926,A -85,B 0,C 180,E1 -18879.241,E2 -18879.241} C_VEL
LIN {X 0,Y 264.157,Z 449.266,A -85,B 0,C 180,E1 -18881.382,E2 -18881.382} C_VEL
LIN {X 0,Y 260.111,Z 452.449,A -85,B 0,C 180,E1 -18884.324,E2 -18884.324} C_VEL
LIN {X 0,Y 256.69,Z 454.325,A -85,B 0,C 180,E1 -18887.348,E2 -18887.348} C_VEL
LIN {X 0,Y 253.952,Z 454.841,A -85,B 0,C 180,E1 -18890.442,E2 -18890.442} C_VEL
LIN {X 0,Y 251.978,Z 453.976,A -85,B 0,C 180,E1 -18893.595,E2 -18893.595} C_VEL
LIN {X 0,Y 251.292,Z 452.979,A -85,B 0,C 180,E1 -18895.187,E2 -18895.187} C_VEL
LIN {X 0,Y 250.516,Z 451.655,A -85,B 0,C 180,E1 -18896.784,E2 -18896.784} C_VEL
LIN {X 0,Y 249.814,Z 448.979,A -85,B 0,C 180,E1 -18899.194,E2 -18899.194} C_VEL
LIN {X 0,Y 249.218,Z 444.004,A -85,B 0,C 180,E1 -18902.425,E2 -18902.425} C_VEL
LIN {X 0,Y 249.076,Z 439.186,A -85,B 0,C 180,E1 -18904.856,E2 -18904.856} C_VEL
LIN {X 0,Y 249.591,Z 432.231,A -85,B 0,C 180,E1 -18907.687,E2 -18907.687} C_VEL
LIN {X 0,Y 250.177,Z 424.67,A -85,B 0,C 180,E1 -18910.206,E2 -18910.206} C_VEL
LIN {X 0,Y 250.913,Z 416.338,A -85,B 0,C 180,E1 -18912.538,E2 -18912.538} C_VEL
LIN {X 0,Y 251.921,Z 406.001,A -85,B 0,C 180,E1 -18914.955,E2 -18914.955} C_VEL
LIN {X 0,Y 253.246,Z 393.602,A -85,B 0,C 180,E1 -18917.358,E2 -18917.358} C_VEL
LIN {X 0,Y 254.633,Z 380.965,A -85,B 0,C 180,E1 -18919.342,E2 -18919.342} C_VEL
LIN {X 0,Y 256.004,Z 367.211,A -85,B 0,C 180,E1 -18921.12,E2 -18921.12} C_VEL
LIN {X 0,Y 256.384,Z 361.844,A -85,B 0,C 180,E1 -18921.72,E2 -18921.72} C_VEL
LIN {X 0,Y 253.362,Z 348.166,A -85,B 0,C 180,E1 -18923.24,E2 -18923.24} C_VEL
LIN {X 0,Y 249.741,Z 332.895,A -85,B 0,C 180,E1 -18924.651,E2 -18924.651} C_VEL
LIN {X 0,Y 248.647,Z 328.14,A -85,B 0,C 180,E1 -18925.047,E2 -18925.047} C_VEL
LIN {X 0,Y 248.737,Z 323.925,A -85,B 0,C 180,E1 -18929.541,E2 -18929.541} C_VEL
LIN {X 0,Y 248.796,Z 323.546,A -85,B 0,C 180,E1 -18930.175,E2 -18930.175} C_VEL
LIN {X 0,Y 249.68,Z 325.159,A -85,B 0,C 180,E1 -18932.387,E2 -18932.387} C_VEL
LIN {X 0,Y 250.631,Z 327.734,A -85,B 0,C 180,E1 -18935.59,E2 -18935.59} C_VEL
LIN {X 0,Y 251.321,Z 330.287,A -85,B 0,C 180,E1 -18938.463,E2 -18938.463} C_VEL
LIN {X 0,Y 251.937,Z 333.665,A -85,B 0,C 180,E1 -18942.029,E2 -18942.029} C_VEL
LIN {X 0,Y 252.575,Z 338.131,A -85,B 0,C 180,E1 -18946.341,E2 -18946.341} C_VEL
LIN {X 0,Y 252.714,Z 338.858,A -85,B 0,C 180,E1 -18946.887,E2 -18946.887} C_VEL
LIN {X 0,Y 254.356,Z 342.102,A -85,B 0,C 180,E1 -18947.362,E2 -18947.362} C_VEL
LIN {X 0,Y 255.592,Z 343.941,A -85,B 0,C 180,E1 -18947.693,E2 -18947.693} C_VEL
LIN {X 0,Y 261.577,Z 355.131,A -85,B 0,C 180,E1 -18949.452,E2 -18949.452} C_VEL
LIN {X 0,Y 267.008,Z 367.474,A -85,B 0,C 180,E1 -18951.313,E2 -18951.313} C_VEL
LIN {X 0,Y 271.636,Z 380.867,A -85,B 0,C 180,E1 -18953.327,E2 -18953.327} C_VEL
LIN {X 0,Y 274.806,Z 393.283,A -85,B 0,C 180,E1 -18955.243,E2 -18955.243} C_VEL
LIN {X 0,Y 275.258,Z 395.536,A -85,B 0,C 180,E1 -18955.604,E2 -18955.604} C_VEL
LIN {X 0,Y 274.774,Z 399.499,A -85,B 0,C 180,E1 -18956.051,E2 -18956.051} C_VEL
LIN {X 0,Y 272.024,Z 412.372,A -85,B 0,C 180,E1 -18957.581,E2 -18957.581} C_VEL
LIN {X 0,Y 268.664,Z 425.101,A -85,B 0,C 180,E1 -18959.416,E2 -18959.416} C_VEL
LIN {X 0,Y 265.398,Z 436.841,A -85,B 0,C 180,E1 -18961.532,E2 -18961.532} C_VEL
LIN {X 0,Y 262.357,Z 446.99,A -85,B 0,C 180,E1 -18963.768,E2 -18963.768} C_VEL
LIN {X 0,Y 259.016,Z 456.91,A -85,B 0,C 180,E1 -18966.408,E2 -18966.408} C_VEL
LIN {X 0,Y 256.162,Z 465.123,A -85,B 0,C 180,E1 -18969.104,E2 -18969.104} C_VEL
LIN {X 0,Y 254.113,Z 471.048,A -85,B 0,C 180,E1 -18971.454,E2 -18971.454} C_VEL
LIN {X 0,Y 251.867,Z 477.512,A -85,B 0,C 180,E1 -18974.628,E2 -18974.628} C_VEL
LIN {X 0,Y 250.191,Z 482.555,A -85,B 0,C 180,E1 -18977.837,E2 -18977.837} C_VEL
LIN {X 0,Y 248.999,Z 486.307,A -85,B 0,C 180,E1 -18981.07,E2 -18981.07} C_VEL
LIN {X 0,Y 248.332,Z 488.292,A -85,B 0,C 180,E1 -18983.5,E2 -18983.5} C_VEL
LIN {X 0,Y 248.087,Z 489.968,A -85,B 0,C 180,E1 -18986.752,E2 -18986.752} C_VEL
LIN {X 0,Y 247.819,Z 490.565,A -85,B 0,C 180,E1 -18990,E2 -18990} C_VEL
LIN {X 0,Y 248.08,Z 490.001,A -85,B 0,C 180,E1 -18993.248,E2 -18993.248} C_VEL
LIN {X 0,Y 248.324,Z 488.369,A -85,B 0,C 180,E1 -18996.5,E2 -18996.5} C_VEL
LIN {X 0,Y 249.228,Z 485.578,A -85,B 0,C 180,E1 -18999.741,E2 -18999.741} C_VEL
LIN {X 0,Y 250.521,Z 481.583,A -85,B 0,C 180,E1 -19002.969,E2 -19002.969} C_VEL
LIN {X 0,Y 252.353,Z 476.26,A -85,B 0,C 180,E1 -19006.17,E2 -19006.17} C_VEL
LIN {X 0,Y 254.748,Z 469.458,A -85,B 0,C 180,E1 -19009.333,E2 -19009.333} C_VEL
LIN {X 0,Y 257.174,Z 462.286,A -85,B 0,C 180,E1 -19012.029,E2 -19012.029} C_VEL
LIN {X 0,Y 260.288,Z 453.343,A -85,B 0,C 180,E1 -19014.74,E2 -19014.74} C_VEL
LIN {X 0,Y 263.808,Z 442.649,A -85,B 0,C 180,E1 -19017.358,E2 -19017.358} C_VEL
LIN {X 0,Y 266.587,Z 432.808,A -85,B 0,C 180,E1 -19019.376,E2 -19019.376} C_VEL
LIN {X 0,Y 270.002,Z 420.757,A -85,B 0,C 180,E1 -19021.371,E2 -19021.371} C_VEL
LIN {X 0,Y 273.18,Z 407.652,A -85,B 0,C 180,E1 -19023.14,E2 -19023.14} C_VEL
LIN {X 0,Y 275.417,Z 396.657,A -85,B 0,C 180,E1 -19024.353,E2 -19024.353} C_VEL
LIN {X 0,Y 273.325,Z 386.655,A -85,B 0,C 180,E1 -19025.909,E2 -19025.909} C_VEL
LIN {X 0,Y 270.147,Z 375.959,A -85,B 0,C 180,E1 -19027.534,E2 -19027.534} C_VEL
LIN {X 0,Y 265.275,Z 363.171,A -85,B 0,C 180,E1 -19029.464,E2 -19029.464} C_VEL
LIN {X 0,Y 259.276,Z 350.503,A -85,B 0,C 180,E1 -19031.4,E2 -19031.4} C_VEL
LIN {X 0,Y 254.634,Z 342.486,A -85,B 0,C 180,E1 -19032.712,E2 -19032.712} C_VEL
LIN {X 0,Y 252.793,Z 339.21,A -85,B 0,C 180,E1 -19033.231,E2 -19033.231} C_VEL
LIN {X 0,Y 252.647,Z 338.757,A -85,B 0,C 180,E1 -19033.292,E2 -19033.292} C_VEL
LIN {X 0,Y 252.196,Z 335.434,A -85,B 0,C 180,E1 -19036.431,E2 -19036.431} C_VEL
LIN {X 0,Y 251.602,Z 331.883,A -85,B 0,C 180,E1 -19040.024,E2 -19040.024} C_VEL
LIN {X 0,Y 250.941,Z 328.309,A -85,B 0,C 180,E1 -19043.975,E2 -19043.975} C_VEL
LIN {X 0,Y 250.28,Z 325.041,A -85,B 0,C 180,E1 -19047.755,E2 -19047.755} C_VEL
LIN {X 0,Y 249.569,Z 322.095,A -85,B 0,C 180,E1 -19051.397,E2 -19051.397} C_VEL
LIN {X 0,Y 249.075,Z 320.067,A -85,B 0,C 180,E1 -19054.153,E2 -19054.153} C_VEL
LIN {X 0,Y 249.089,Z 320.062,A -85,B 0,C 180,E1 -19058.605,E2 -19058.605} C_VEL
LIN {X 0,Y 249.196,Z 320.047,A -85,B 0,C 180,E1 -19063.619,E2 -19063.619} C_VEL
LIN {X 0,Y 249.234,Z 320.039,A -85,B 0,C 180,E1 -19068.615,E2 -19068.615} C_VEL
LIN {X 0,Y 249.435,Z 320.032,A -85,B 0,C 180,E1 -19071.901,E2 -19071.901} C_VEL
LIN {X 0,Y 249.28,Z 320.038,A -85,B 0,C 180,E1 -19075.148,E2 -19075.148} C_VEL
LIN {X 0,Y 249.675,Z 319.989,A -85,B 0,C 180,E1 -19078.387,E2 -19078.387} C_VEL
LIN {X 0,Y 249.671,Z 320,A -85,B 0,C 180,E1 -19081.613,E2 -19081.613} C_VEL
LIN {X 0,Y 249.437,Z 320.017,A -85,B 0,C 180,E1 -19086.471,E2 -19086.471} C_VEL
LIN {X 0,Y 249.342,Z 320.031,A -85,B 0,C 180,E1 -19089.736,E2 -19089.736} C_VEL
LIN {X 0,Y 249.206,Z 320.057,A -85,B 0,C 180,E1 -19094.703,E2 -19094.703} C_VEL
LIN {X 0,Y 249.139,Z 320.063,A -85,B 0,C 180,E1 -19098.077,E2 -19098.077} C_VEL
LIN {X 0,Y 249.083,Z 320.06,A -85,B 0,C 180,E1 -19101.518,E2 -19101.518} C_VEL
LIN {X 0,Y 249.068,Z 320.072,A -85,B 0,C 180,E1 -19104.609,E2 -19104.609} C_VEL
LIN {X 0,Y 248.628,Z 320.633,A -85,B 0,C 180,E1 -19105.956,E2 -19105.956} C_VEL
LIN {X 0,Y 247.494,Z 322.067,A -85,B 0,C 180,E1 -19107.263,E2 -19107.263} C_VEL
LIN {X 0,Y 244.97,Z 326.368,A -85,B 0,C 180,E1 -19109.822,E2 -19109.822} C_VEL
LIN {X 0,Y 244.498,Z 328.692,A -85,B 0,C 180,E1 -19111.124,E2 -19111.124} C_VEL
LIN {X 0,Y 244.579,Z 329.423,A -85,B 0,C 180,E1 -19111.563,E2 -19111.563} C_VEL
LIN {X 0,Y 245.969,Z 335.527,A -85,B 0,C 180,E1 -19114.851,E2 -19114.851} C_VEL
LIN {X 0,Y 248.276,Z 344.319,A -85,B 0,C 180,E1 -19119.045,E2 -19119.045} C_VEL
LIN {X 0,Y 250.928,Z 354.898,A -85,B 0,C 180,E1 -19123.264,E2 -19123.264} C_VEL
LIN {X 0,Y 252.818,Z 362.326,A -85,B 0,C 180,E1 -19125.976,E2 -19125.976} C_VEL
LIN {X 0,Y 253.635,Z 365.504,A -85,B 0,C 180,E1 -19127.028,E2 -19127.028} C_VEL
LIN {X 0,Y 258.86,Z 375.612,A -85,B 0,C 180,E1 -19128.445,E2 -19128.445} C_VEL
LIN {X 0,Y 262.099,Z 392.095,A -85,B 0,C 180,E1 -19129.831,E2 -19129.831} C_VEL
LIN {X 0,Y 263.565,Z 404.41,A -85,B 0,C 180,E1 -19130.945,E2 -19130.945} C_VEL
LIN {X 0,Y 264.268,Z 419.729,A -85,B 0,C 180,E1 -19132.459,E2 -19132.459} C_VEL
LIN {X 0,Y 264.011,Z 434.574,A -85,B 0,C 180,E1 -19134.152,E2 -19134.152} C_VEL
LIN {X 0,Y 263.228,Z 446.184,A -85,B 0,C 180,E1 -19135.666,E2 -19135.666} C_VEL
LIN {X 0,Y 259.697,Z 459.633,A -85,B 0,C 180,E1 -19137.462,E2 -19137.462} C_VEL
LIN {X 0,Y 255.977,Z 471.866,A -85,B 0,C 180,E1 -19139.474,E2 -19139.474} C_VEL
LIN {X 0,Y 252.419,Z 483.058,A -85,B 0,C 180,E1 -19141.75,E2 -19141.75} C_VEL
LIN {X 0,Y 249.302,Z 492.824,A -85,B 0,C 180,E1 -19144.18,E2 -19144.18} C_VEL
LIN {X 0,Y 246.422,Z 501.83,A -85,B 0,C 180,E1 -19146.912,E2 -19146.912} C_VEL
LIN {X 0,Y 244.025,Z 509.579,A -85,B 0,C 180,E1 -19149.782,E2 -19149.782} C_VEL
LIN {X 0,Y 242.053,Z 516.852,A -85,B 0,C 180,E1 -19153.122,E2 -19153.122} C_VEL
LIN {X 0,Y 240.83,Z 522.602,A -85,B 0,C 180,E1 -19156.5,E2 -19156.5} C_VEL
LIN {X 0,Y 240.292,Z 526.977,A -85,B 0,C 180,E1 -19159.893,E2 -19159.893} C_VEL
LIN {X 0,Y 240.417,Z 530.357,A -85,B 0,C 180,E1 -19163.671,E2 -19163.671} C_VEL
LIN {X 0,Y 240.511,Z 531.94,A -85,B 0,C 180,E1 -19166.65,E2 -19166.65} C_VEL
LIN {X 0,Y 240.75,Z 532.428,A -85,B 0,C 180,E1 -19168.328,E2 -19168.328} C_VEL
LIN {X 0,Y 240.839,Z 532.596,A -85,B 0,C 180,E1 -19170,E2 -19170} C_VEL
LIN {X 0,Y 240.789,Z 532.429,A -85,B 0,C 180,E1 -19171.673,E2 -19171.673} C_VEL
LIN {X 0,Y 240.493,Z 531.157,A -85,B 0,C 180,E1 -19175.03,E2 -19175.03} C_VEL
LIN {X 0,Y 240.273,Z 528.66,A -85,B 0,C 180,E1 -19178.41,E2 -19178.41} C_VEL
LIN {X 0,Y 240.479,Z 524.91,A -85,B 0,C 180,E1 -19181.805,E2 -19181.805} C_VEL
LIN {X 0,Y 241.394,Z 519.85,A -85,B 0,C 180,E1 -19185.191,E2 -19185.191} C_VEL
LIN {X 0,Y 242.938,Z 513.345,A -85,B 0,C 180,E1 -19188.556,E2 -19188.556} C_VEL
LIN {X 0,Y 245.375,Z 505.229,A -85,B 0,C 180,E1 -19191.861,E2 -19191.861} C_VEL
LIN {X 0,Y 248.12,Z 496.596,A -85,B 0,C 180,E1 -19194.696,E2 -19194.696} C_VEL
LIN {X 0,Y 249.92,Z 491.23,A -85,B 0,C 180,E1 -19196.289,E2 -19196.289} C_VEL
LIN {X 0,Y 255.209,Z 482.161,A -85,B 0,C 180,E1 -19199.716,E2 -19199.716} C_VEL
LIN {X 0,Y 260.954,Z 472.779,A -85,B 0,C 180,E1 -19202.592,E2 -19202.592} C_VEL
LIN {X 0,Y 268.465,Z 460.87,A -85,B 0,C 180,E1 -19205.485,E2 -19205.485} C_VEL
LIN {X 0,Y 274.42,Z 450.967,A -85,B 0,C 180,E1 -19207.509,E2 -19207.509} C_VEL
LIN {X 0,Y 280.752,Z 437.993,A -85,B 0,C 180,E1 -19210.136,E2 -19210.136} C_VEL
LIN {X 0,Y 284.564,Z 428.27,A -85,B 0,C 180,E1 -19212.299,E2 -19212.299} C_VEL
LIN {X 0,Y 287.725,Z 419.642,A -85,B 0,C 180,E1 -19214.436,E2 -19214.436} C_VEL
LIN {X 0,Y 287.733,Z 418.409,A -85,B 0,C 180,E1 -19215.1,E2 -19215.1} C_VEL
LIN {X 0,Y 287.161,Z 415.911,A -85,B 0,C 180,E1 -19217.242,E2 -19217.242} C_VEL
LIN {X 0,Y 286.903,Z 414.3,A -85,B 0,C 180,E1 -19219.41,E2 -19219.41} C_VEL
LIN {X 0,Y 286.831,Z 413.754,A -85,B 0,C 180,E1 -19221.636,E2 -19221.636} C_VEL
LIN {X 0,Y 286.785,Z 414.405,A -85,B 0,C 180,E1 -19223.974,E2 -19223.974} C_VEL
LIN {X 0,Y 286.708,Z 416.486,A -85,B 0,C 180,E1 -19226.454,E2 -19226.454} C_VEL
LIN {X 0,Y 286.489,Z 418.609,A -85,B 0,C 180,E1 -19228.106,E2 -19228.106} C_VEL
LIN {X 0,Y 285.495,Z 420.576,A -85,B 0,C 180,E1 -19228.872,E2 -19228.872} C_VEL
LIN {X 0,Y 278.185,Z 430.333,A -85,B 0,C 180,E1 -19231.314,E2 -19231.314} C_VEL
LIN {X 0,Y 271.547,Z 438.27,A -85,B 0,C 180,E1 -19233.897,E2 -19233.897} C_VEL
LIN {X 0,Y 265.518,Z 444.675,A -85,B 0,C 180,E1 -19236.607,E2 -19236.607} C_VEL
LIN {X 0,Y 260.183,Z 449.579,A -85,B 0,C 180,E1 -19239.442,E2 -19239.442} C_VEL
LIN {X 0,Y 255.551,Z 453.117,A -85,B 0,C 180,E1 -19242.391,E2 -19242.391} C_VEL
LIN {X 0,Y 251.68,Z 455.336,A -85,B 0,C 180,E1 -19245.445,E2 -19245.445} C_VEL
LIN {X 0,Y 248.425,Z 456.256,A -85,B 0,C 180,E1 -19248.578,E2 -19248.578} C_VEL
LIN {X 0,Y 245.975,Z 455.774,A -85,B 0,C 180,E1 -19251.787,E2 -19251.787} C_VEL
LIN {X 0,Y 244.304,Z 453.899,A -85,B 0,C 180,E1 -19255.049,E2 -19255.049} C_VEL
LIN {X 0,Y 243.489,Z 452.458,A -85,B 0,C 180,E1 -19256.691,E2 -19256.691} C_VEL
LIN {X 0,Y 242.745,Z 449.565,A -85,B 0,C 180,E1 -19259.171,E2 -19259.171} C_VEL
LIN {X 0,Y 242.14,Z 444.365,A -85,B 0,C 180,E1 -19262.495,E2 -19262.495} C_VEL
LIN {X 0,Y 242.025,Z 439.325,A -85,B 0,C 180,E1 -19264.998,E2 -19264.998} C_VEL
LIN {X 0,Y 242.543,Z 432.149,A -85,B 0,C 180,E1 -19267.911,E2 -19267.911} C_VEL
LIN {X 0,Y 243.207,Z 423.592,A -85,B 0,C 180,E1 -19270.73,E2 -19270.73} C_VEL
LIN {X 0,Y 244.101,Z 414.079,A -85,B 0,C 180,E1 -19273.317,E2 -19273.317} C_VEL
LIN {X 0,Y 245.199,Z 403.1,A -85,B 0,C 180,E1 -19275.801,E2 -19275.801} C_VEL
LIN {X 0,Y 246.671,Z 389.827,A -85,B 0,C 180,E1 -19278.265,E2 -19278.265} C_VEL
LIN {X 0,Y 248.126,Z 376.901,A -85,B 0,C 180,E1 -19280.221,E2 -19280.221} C_VEL
LIN {X 0,Y 249.423,Z 363.282,A -85,B 0,C 180,E1 -19281.913,E2 -19281.913} C_VEL
LIN {X 0,Y 246.579,Z 350.034,A -85,B 0,C 180,E1 -19283.441,E2 -19283.441} C_VEL
LIN {X 0,Y 242.79,Z 333.996,A -85,B 0,C 180,E1 -19284.972,E2 -19284.972} C_VEL
LIN {X 0,Y 241.617,Z 328.754,A -85,B 0,C 180,E1 -19285.424,E2 -19285.424} C_VEL
LIN {X 0,Y 241.737,Z 325.533,A -85,B 0,C 180,E1 -19289.099,E2 -19289.099} C_VEL
LIN {X 0,Y 243.29,Z 328.295,A -85,B 0,C 180,E1 -19293.098,E2 -19293.098} C_VEL
LIN {X 0,Y 244.171,Z 330.851,A -85,B 0,C 180,E1 -19296.299,E2 -19296.299} C_VEL
LIN {X 0,Y 244.754,Z 333.386,A -85,B 0,C 180,E1 -19299.177,E2 -19299.177} C_VEL
LIN {X 0,Y 245.225,Z 335.867,A -85,B 0,C 180,E1 -19301.828,E2 -19301.828} C_VEL
LIN {X 0,Y 245.806,Z 339.625,A -85,B 0,C 180,E1 -19305.364,E2 -19305.364} C_VEL
LIN {X 0,Y 247.566,Z 342.847,A -85,B 0,C 180,E1 -19305.901,E2 -19305.901} C_VEL
LIN {X 0,Y 248.814,Z 344.508,A -85,B 0,C 180,E1 -19306.251,E2 -19306.251} C_VEL
LIN {X 0,Y 254.263,Z 354.252,A -85,B 0,C 180,E1 -19307.924,E2 -19307.924} C_VEL
LIN {X 0,Y 259.438,Z 365.315,A -85,B 0,C 180,E1 -19309.725,E2 -19309.725} C_VEL
LIN {X 0,Y 263.697,Z 376.665,A -85,B 0,C 180,E1 -19311.527,E2 -19311.527} C_VEL
LIN {X 0,Y 267.135,Z 388.16,A -85,B 0,C 180,E1 -19313.362,E2 -19313.362} C_VEL
LIN {X 0,Y 269.248,Z 397.825,A -85,B 0,C 180,E1 -19314.952,E2 -19314.952} C_VEL
LIN {X 0,Y 266.776,Z 410.198,A -85,B 0,C 180,E1 -19316.411,E2 -19316.411} C_VEL
LIN {X 0,Y 263.429,Z 422.956,A -85,B 0,C 180,E1 -19318.203,E2 -19318.203} C_VEL
LIN {X 0,Y 260.427,Z 433.42,A -85,B 0,C 180,E1 -19319.995,E2 -19319.995} C_VEL
LIN {X 0,Y 257.112,Z 444.43,A -85,B 0,C 180,E1 -19322.31,E2 -19322.31} C_VEL
LIN {X 0,Y 253.945,Z 453.518,A -85,B 0,C 180,E1 -19324.598,E2 -19324.598} C_VEL
LIN {X 0,Y 250.754,Z 462.417,A -85,B 0,C 180,E1 -19327.333,E2 -19327.333} C_VEL
LIN {X 0,Y 248.128,Z 469.777,A -85,B 0,C 180,E1 -19330.129,E2 -19330.129} C_VEL
LIN {X 0,Y 246.115,Z 475.081,A -85,B 0,C 180,E1 -19332.552,E2 -19332.552} C_VEL
LIN {X 0,Y 244.081,Z 480.811,A -85,B 0,C 180,E1 -19335.833,E2 -19335.833} C_VEL
LIN {X 0,Y 242.899,Z 484.189,A -85,B 0,C 180,E1 -19338.314,E2 -19338.314} C_VEL
LIN {X 0,Y 241.722,Z 487.627,A -85,B 0,C 180,E1 -19341.641,E2 -19341.641} C_VEL
LIN {X 0,Y 241.181,Z 489.872,A -85,B 0,C 180,E1 -19344.984,E2 -19344.984} C_VEL
LIN {X 0,Y 240.839,Z 491.018,A -85,B 0,C 180,E1 -19348.327,E2 -19348.327} C_VEL
LIN {X 0,Y 240.838,Z 491.028,A -85,B 0,C 180,E1 -19351.672,E2 -19351.672} C_VEL
LIN {X 0,Y 241.159,Z 489.927,A -85,B 0,C 180,E1 -19355.015,E2 -19355.015} C_VEL
LIN {X 0,Y 241.776,Z 487.722,A -85,B 0,C 180,E1 -19358.357,E2 -19358.357} C_VEL
LIN {X 0,Y 242.891,Z 484.344,A -85,B 0,C 180,E1 -19361.685,E2 -19361.685} C_VEL
LIN {X 0,Y 244.488,Z 479.706,A -85,B 0,C 180,E1 -19364.993,E2 -19364.993} C_VEL
LIN {X 0,Y 246.654,Z 473.669,A -85,B 0,C 180,E1 -19368.266,E2 -19368.266} C_VEL
LIN {X 0,Y 249.232,Z 466.654,A -85,B 0,C 180,E1 -19371.264,E2 -19371.264} C_VEL
LIN {X 0,Y 252.45,Z 457.909,A -85,B 0,C 180,E1 -19374.244,E2 -19374.244} C_VEL
LIN {X 0,Y 255.92,Z 448.067,A -85,B 0,C 180,E1 -19376.944,E2 -19376.944} C_VEL
LIN {X 0,Y 259.033,Z 438.014,A -85,B 0,C 180,E1 -19379.233,E2 -19379.233} C_VEL
LIN {X 0,Y 262.382,Z 427.049,A -85,B 0,C 180,E1 -19381.263,E2 -19381.263} C_VEL
LIN {X 0,Y 265.928,Z 413.792,A -85,B 0,C 180,E1 -19383.256,E2 -19383.256} C_VEL
LIN {X 0,Y 269.019,Z 400.333,A -85,B 0,C 180,E1 -19384.876,E2 -19384.876} C_VEL
LIN {X 0,Y 269.272,Z 397.687,A -85,B 0,C 180,E1 -19385.195,E2 -19385.195} C_VEL
LIN {X 0,Y 266.538,Z 385.65,A -85,B 0,C 180,E1 -19387.159,E2 -19387.159} C_VEL
LIN {X 0,Y 262.509,Z 373.069,A -85,B 0,C 180,E1 -19389.179,E2 -19389.179} C_VEL
LIN {X 0,Y 257.54,Z 360.883,A -85,B 0,C 180,E1 -19391.125,E2 -19391.125} C_VEL
LIN {X 0,Y 252.062,Z 350.258,A -85,B 0,C 180,E1 -19392.908,E2 -19392.908} C_VEL
LIN {X 0,Y 248.188,Z 343.638,A -85,B 0,C 180,E1 -19394.078,E2 -19394.078} C_VEL
LIN {X 0,Y 246.156,Z 340.697,A -85,B 0,C 180,E1 -19394.665,E2 -19394.665} C_VEL
LIN {X 0,Y 245.694,Z 339.454,A -85,B 0,C 180,E1 -19394.868,E2 -19394.868} C_VEL
LIN {X 0,Y 245.19,Z 335.493,A -85,B 0,C 180,E1 -19398.756,E2 -19398.756} C_VEL
LIN {X 0,Y 244.341,Z 331.123,A -85,B 0,C 180,E1 -19403.645,E2 -19403.645} C_VEL
LIN {X 0,Y 243.808,Z 328.444,A -85,B 0,C 180,E1 -19406.791,E2 -19406.791} C_VEL
LIN {X 0,Y 243.153,Z 325.494,A -85,B 0,C 180,E1 -19410.57,E2 -19410.57} C_VEL
LIN {X 0,Y 242.495,Z 322.72,A -85,B 0,C 180,E1 -19414.232,E2 -19414.232} C_VEL
LIN {X 0,Y 242.017,Z 320.951,A -85,B 0,C 180,E1 -19416.919,E2 -19416.919} C_VEL
LIN {X 0,Y 242.054,Z 320.95,A -85,B 0,C 180,E1 -19421.374,E2 -19421.374} C_VEL
LIN {X 0,Y 242.14,Z 320.937,A -85,B 0,C 180,E1 -19424.857,E2 -19424.857} C_VEL
LIN {X 0,Y 242.329,Z 320.917,A -85,B 0,C 180,E1 -19430.421,E2 -19430.421} C_VEL
LIN {X 0,Y 242.403,Z 320.889,A -85,B 0,C 180,E1 -19433.34,E2 -19433.34} C_VEL
LIN {X 0,Y 242.635,Z 320.866,A -85,B 0,C 180,E1 -19438.34,E2 -19438.34} C_VEL
LIN {X 0,Y 242.631,Z 320.877,A -85,B 0,C 180,E1 -19441.66,E2 -19441.66} C_VEL
LIN {X 0,Y 242.408,Z 320.894,A -85,B 0,C 180,E1 -19446.659,E2 -19446.659} C_VEL
LIN {X 0,Y 242.266,Z 320.909,A -85,B 0,C 180,E1 -19450.024,E2 -19450.024} C_VEL
LIN {X 0,Y 242.167,Z 320.926,A -85,B 0,C 180,E1 -19455.141,E2 -19455.141} C_VEL
LIN {X 0,Y 242.073,Z 320.952,A -85,B 0,C 180,E1 -19458.624,E2 -19458.624} C_VEL
LIN {X 0,Y 242.004,Z 320.943,A -85,B 0,C 180,E1 -19462.181,E2 -19462.181} C_VEL
LIN {X 0,Y 242.065,Z 321.078,A -85,B 0,C 180,E1 -19465.499,E2 -19465.499} C_VEL
LIN {X 0,Y 242.954,Z 323.695,A -85,B 0,C 180,E1 -19467.57,E2 -19467.57} C_VEL
LIN {X 0,Y 243.599,Z 324.592,A -85,B 0,C 180,E1 -19468.427,E2 -19468.427} C_VEL
LIN {X 0,Y 244.579,Z 329.423,A -85,B 0,C 180,E1 -19471.563,E2 -19471.563} C_VEL
LIN {X 0,Y 244.646,Z 331.065,A -85,B 0,C 180,E1 -19472.405,E2 -19472.405} C_VEL
LIN {X 0,Y 243.792,Z 335.238,A -85,B 0,C 180,E1 -19473.979,E2 -19473.979} C_VEL
LIN {X 0,Y 241.952,Z 342.027,A -85,B 0,C 180,E1 -19476.255,E2 -19476.255} C_VEL
LIN {X 0,Y 241.738,Z 345.167,A -85,B 0,C 180,E1 -19477.452,E2 -19477.452} C_VEL
LIN {X 0,Y 241.887,Z 346.106,A -85,B 0,C 180,E1 -19477.864,E2 -19477.864} C_VEL
LIN {X 0,Y 244.221,Z 355.73,A -85,B 0,C 180,E1 -19481.995,E2 -19481.995} C_VEL
LIN {X 0,Y 246.49,Z 364.917,A -85,B 0,C 180,E1 -19485.464,E2 -19485.464} C_VEL
LIN {X 0,Y 249.063,Z 369.731,A -85,B 0,C 180,E1 -19486.22,E2 -19486.22} C_VEL
LIN {X 0,Y 253.906,Z 379.214,A -85,B 0,C 180,E1 -19487.614,E2 -19487.614} C_VEL
LIN {X 0,Y 256.707,Z 395.18,A -85,B 0,C 180,E1 -19489.046,E2 -19489.046} C_VEL
LIN {X 0,Y 257.944,Z 407.961,A -85,B 0,C 180,E1 -19490.268,E2 -19490.268} C_VEL
LIN {X 0,Y 258.372,Z 423.084,A -85,B 0,C 180,E1 -19491.878,E2 -19491.878} C_VEL
LIN {X 0,Y 257.793,Z 437.544,A -85,B 0,C 180,E1 -19493.634,E2 -19493.634} C_VEL
LIN {X 0,Y 256.975,Z 447.019,A -85,B 0,C 180,E1 -19494.948,E2 -19494.948} C_VEL
LIN {X 0,Y 253.318,Z 460.209,A -85,B 0,C 180,E1 -19496.775,E2 -19496.775} C_VEL
LIN {X 0,Y 249.86,Z 471.264,A -85,B 0,C 180,E1 -19498.644,E2 -19498.644} C_VEL
LIN {X 0,Y 246.089,Z 482.446,A -85,B 0,C 180,E1 -19500.955,E2 -19500.955} C_VEL
LIN {X 0,Y 242.939,Z 491.91,A -85,B 0,C 180,E1 -19503.359,E2 -19503.359} C_VEL
LIN {X 0,Y 239.785,Z 501.213,A -85,B 0,C 180,E1 -19506.234,E2 -19506.234} C_VEL
LIN {X 0,Y 237.268,Z 508.962,A -85,B 0,C 180,E1 -19509.18,E2 -19509.18} C_VEL
LIN {X 0,Y 235.178,Z 516.235,A -85,B 0,C 180,E1 -19512.613,E2 -19512.613} C_VEL
LIN {X 0,Y 233.844,Z 521.986,A -85,B 0,C 180,E1 -19516.088,E2 -19516.088} C_VEL
LIN {X 0,Y 233.23,Z 526.36,A -85,B 0,C 180,E1 -19519.584,E2 -19519.584} C_VEL
LIN {X 0,Y 233.25,Z 529.465,A -85,B 0,C 180,E1 -19523.078,E2 -19523.078} C_VEL
LIN {X 0,Y 233.387,Z 530.555,A -85,B 0,C 180,E1 -19524.817,E2 -19524.817} C_VEL
LIN {X 0,Y 233.667,Z 531.819,A -85,B 0,C 180,E1 -19528.277,E2 -19528.277} C_VEL
LIN {X 0,Y 233.782,Z 531.989,A -85,B 0,C 180,E1 -19530,E2 -19530} C_VEL
LIN {X 0,Y 233.704,Z 531.819,A -85,B 0,C 180,E1 -19531.724,E2 -19531.724} C_VEL
LIN {X 0,Y 233.401,Z 530.544,A -85,B 0,C 180,E1 -19535.183,E2 -19535.183} C_VEL
LIN {X 0,Y 233.191,Z 528.043,A -85,B 0,C 180,E1 -19538.667,E2 -19538.667} C_VEL
LIN {X 0,Y 233.442,Z 524.291,A -85,B 0,C 180,E1 -19542.166,E2 -19542.166} C_VEL
LIN {X 0,Y 234.438,Z 519.229,A -85,B 0,C 180,E1 -19545.653,E2 -19545.653} C_VEL
LIN {X 0,Y 236.117,Z 512.726,A -85,B 0,C 180,E1 -19549.112,E2 -19549.112} C_VEL
LIN {X 0,Y 238.322,Z 505.748,A -85,B 0,C 180,E1 -19552.086,E2 -19552.086} C_VEL
LIN {X 0,Y 241.108,Z 497.534,A -85,B 0,C 180,E1 -19554.937,E2 -19554.937} C_VEL
LIN {X 0,Y 242.716,Z 492.624,A -85,B 0,C 180,E1 -19556.436,E2 -19556.436} C_VEL
LIN {X 0,Y 248.398,Z 483.679,A -85,B 0,C 180,E1 -19560.147,E2 -19560.147} C_VEL
LIN {X 0,Y 255.057,Z 473.698,A -85,B 0,C 180,E1 -19563.443,E2 -19563.443} C_VEL
LIN {X 0,Y 263.106,Z 462.026,A -85,B 0,C 180,E1 -19566.457,E2 -19566.457} C_VEL
LIN {X 0,Y 269.147,Z 452.802,A -85,B 0,C 180,E1 -19568.431,E2 -19568.431} C_VEL
LIN {X 0,Y 275.783,Z 440.739,A -85,B 0,C 180,E1 -19571.012,E2 -19571.012} C_VEL
LIN {X 0,Y 280.33,Z 430.817,A -85,B 0,C 180,E1 -19573.361,E2 -19573.361} C_VEL
LIN {X 0,Y 282.87,Z 424.917,A -85,B 0,C 180,E1 -19574.885,E2 -19574.885} C_VEL
LIN {X 0,Y 283.176,Z 423.622,A -85,B 0,C 180,E1 -19575.426,E2 -19575.426} C_VEL
LIN {X 0,Y 282.627,Z 420.693,A -85,B 0,C 180,E1 -19578.246,E2 -19578.246} C_VEL
LIN {X 0,Y 282.441,Z 419.456,A -85,B 0,C 180,E1 -19580.478,E2 -19580.478} C_VEL
LIN {X 0,Y 282.257,Z 419.491,A -85,B 0,C 180,E1 -19582.824,E2 -19582.824} C_VEL
LIN {X 0,Y 282.055,Z 420.739,A -85,B 0,C 180,E1 -19585.313,E2 -19585.313} C_VEL
LIN {X 0,Y 281.778,Z 422.083,A -85,B 0,C 180,E1 -19586.721,E2 -19586.721} C_VEL
LIN {X 0,Y 281.465,Z 423.246,A -85,B 0,C 180,E1 -19587.648,E2 -19587.648} C_VEL
LIN {X 0,Y 280.202,Z 425.05,A -85,B 0,C 180,E1 -19588.216,E2 -19588.216} C_VEL
LIN {X 0,Y 272.62,Z 434.173,A -85,B 0,C 180,E1 -19590.672,E2 -19590.672} C_VEL
LIN {X 0,Y 265.768,Z 441.526,A -85,B 0,C 180,E1 -19593.285,E2 -19593.285} C_VEL
LIN {X 0,Y 259.468,Z 447.455,A -85,B 0,C 180,E1 -19596.028,E2 -19596.028} C_VEL
LIN {X 0,Y 253.919,Z 452.012,A -85,B 0,C 180,E1 -19598.911,E2 -19598.911} C_VEL
LIN {X 0,Y 249.108,Z 455.215,A -85,B 0,C 180,E1 -19601.921,E2 -19601.921} C_VEL
LIN {X 0,Y 245.025,Z 457.074,A -85,B 0,C 180,E1 -19605.04,E2 -19605.04} C_VEL
LIN {X 0,Y 241.622,Z 457.669,A -85,B 0,C 180,E1 -19608.252,E2 -19608.252} C_VEL
LIN {X 0,Y 239.058,Z 456.927,A -85,B 0,C 180,E1 -19611.547,E2 -19611.547} C_VEL
LIN {X 0,Y 237.315,Z 454.797,A -85,B 0,C 180,E1 -19614.903,E2 -19614.903} C_VEL
LIN {X 0,Y 236.443,Z 453.223,A -85,B 0,C 180,E1 -19616.592,E2 -19616.592} C_VEL
LIN {X 0,Y 235.678,Z 450.116,A -85,B 0,C 180,E1 -19619.146,E2 -19619.146} C_VEL
LIN {X 0,Y 235.164,Z 446.149,A -85,B 0,C 180,E1 -19621.713,E2 -19621.713} C_VEL
LIN {X 0,Y 234.916,Z 441.258,A -85,B 0,C 180,E1 -19624.29,E2 -19624.29} C_VEL
LIN {X 0,Y 235.335,Z 434.217,A -85,B 0,C 180,E1 -19627.292,E2 -19627.292} C_VEL
LIN {X 0,Y 235.995,Z 425.587,A -85,B 0,C 180,E1 -19630.293,E2 -19630.293} C_VEL
LIN {X 0,Y 236.815,Z 416.673,A -85,B 0,C 180,E1 -19632.861,E2 -19632.861} C_VEL
LIN {X 0,Y 237.867,Z 406.031,A -85,B 0,C 180,E1 -19635.421,E2 -19635.421} C_VEL
LIN {X 0,Y 239.136,Z 394.334,A -85,B 0,C 180,E1 -19637.753,E2 -19637.753} C_VEL
LIN {X 0,Y 240.621,Z 381.595,A -85,B 0,C 180,E1 -19639.849,E2 -19639.849} C_VEL
LIN {X 0,Y 242.077,Z 367.791,A -85,B 0,C 180,E1 -19641.715,E2 -19641.715} C_VEL
LIN {X 0,Y 242.418,Z 364.177,A -85,B 0,C 180,E1 -19642.141,E2 -19642.141} C_VEL
LIN {X 0,Y 239.408,Z 350.497,A -85,B 0,C 180,E1 -19643.771,E2 -19643.771} C_VEL
LIN {X 0,Y 235.786,Z 334.797,A -85,B 0,C 180,E1 -19645.32,E2 -19645.32} C_VEL
LIN {X 0,Y 234.567,Z 329.383,A -85,B 0,C 180,E1 -19645.81,E2 -19645.81} C_VEL
LIN {X 0,Y 234.638,Z 327.566,A -85,B 0,C 180,E1 -19647.905,E2 -19647.905} C_VEL
LIN {X 0,Y 235.7,Z 329.141,A -85,B 0,C 180,E1 -19650.458,E2 -19650.458} C_VEL
LIN {X 0,Y 236.883,Z 331.485,A -85,B 0,C 180,E1 -19653.826,E2 -19653.826} C_VEL
LIN {X 0,Y 237.717,Z 334.032,A -85,B 0,C 180,E1 -19657.036,E2 -19657.036} C_VEL
LIN {X 0,Y 238.541,Z 338.018,A -85,B 0,C 180,E1 -19661.5,E2 -19661.5} C_VEL
LIN {X 0,Y 238.828,Z 340.183,A -85,B 0,C 180,E1 -19663.679,E2 -19663.679} C_VEL
LIN {X 0,Y 240.603,Z 343.481,A -85,B 0,C 180,E1 -19664.268,E2 -19664.268} C_VEL
LIN {X 0,Y 242.148,Z 345.486,A -85,B 0,C 180,E1 -19664.735,E2 -19664.735} C_VEL
LIN {X 0,Y 247.49,Z 354.41,A -85,B 0,C 180,E1 -19666.455,E2 -19666.455} C_VEL
LIN {X 0,Y 252.629,Z 365.109,A -85,B 0,C 180,E1 -19668.332,E2 -19668.332} C_VEL
LIN {X 0,Y 256.683,Z 375.305,A -85,B 0,C 180,E1 -19670.054,E2 -19670.054} C_VEL
LIN {X 0,Y 260.218,Z 386.609,A -85,B 0,C 180,E1 -19671.955,E2 -19671.955} C_VEL
LIN {X 0,Y 262.949,Z 398.476,A -85,B 0,C 180,E1 -19673.984,E2 -19673.984} C_VEL
LIN {X 0,Y 263.193,Z 400.577,A -85,B 0,C 180,E1 -19674.322,E2 -19674.322} C_VEL
LIN {X 0,Y 260.212,Z 413.568,A -85,B 0,C 180,E1 -19675.914,E2 -19675.914} C_VEL
LIN {X 0,Y 256.773,Z 425.842,A -85,B 0,C 180,E1 -19677.742,E2 -19677.742} C_VEL
LIN {X 0,Y 253.497,Z 436.729,A -85,B 0,C 180,E1 -19679.745,E2 -19679.745} C_VEL
LIN {X 0,Y 250.306,Z 446.618,A -85,B 0,C 180,E1 -19681.946,E2 -19681.946} C_VEL
LIN {X 0,Y 247.088,Z 455.494,A -85,B 0,C 180,E1 -19684.293,E2 -19684.293} C_VEL
LIN {X 0,Y 243.717,Z 464.393,A -85,B 0,C 180,E1 -19687.179,E2 -19687.179} C_VEL
LIN {X 0,Y 240.707,Z 472.267,A -85,B 0,C 180,E1 -19690.38,E2 -19690.38} C_VEL
LIN {X 0,Y 238.237,Z 478.731,A -85,B 0,C 180,E1 -19693.724,E2 -19693.724} C_VEL
LIN {X 0,Y 236.341,Z 483.776,A -85,B 0,C 180,E1 -19697.113,E2 -19697.113} C_VEL
LIN {X 0,Y 234.925,Z 487.78,A -85,B 0,C 180,E1 -19700.833,E2 -19700.833} C_VEL
LIN {X 0,Y 234.118,Z 490.482,A -85,B 0,C 180,E1 -19704.833,E2 -19704.833} C_VEL
LIN {X 0,Y 234.003,Z 491.182,A -85,B 0,C 180,E1 -19706.556,E2 -19706.556} C_VEL
LIN {X 0,Y 233.716,Z 491.778,A -85,B 0,C 180,E1 -19710,E2 -19710} C_VEL
LIN {X 0,Y 233.995,Z 491.214,A -85,B 0,C 180,E1 -19713.443,E2 -19713.443} C_VEL
LIN {X 0,Y 234.278,Z 489.584,A -85,B 0,C 180,E1 -19716.891,E2 -19716.891} C_VEL
LIN {X 0,Y 235.284,Z 486.794,A -85,B 0,C 180,E1 -19720.324,E2 -19720.324} C_VEL
LIN {X 0,Y 236.721,Z 482.799,A -85,B 0,C 180,E1 -19723.739,E2 -19723.739} C_VEL
LIN {X 0,Y 238.755,Z 477.475,A -85,B 0,C 180,E1 -19727.119,E2 -19727.119} C_VEL
LIN {X 0,Y 241.415,Z 470.67,A -85,B 0,C 180,E1 -19730.447,E2 -19730.447} C_VEL
LIN {X 0,Y 244.079,Z 463.496,A -85,B 0,C 180,E1 -19733.278,E2 -19733.278} C_VEL
LIN {X 0,Y 247.493,Z 454.548,A -85,B 0,C 180,E1 -19736.113,E2 -19736.113} C_VEL
LIN {X 0,Y 251.309,Z 443.849,A -85,B 0,C 180,E1 -19738.842,E2 -19738.842} C_VEL
LIN {X 0,Y 254.542,Z 433.417,A -85,B 0,C 180,E1 -19741.052,E2 -19741.052} C_VEL
LIN {X 0,Y 258.374,Z 420.732,A -85,B 0,C 180,E1 -19743.19,E2 -19743.19} C_VEL
LIN {X 0,Y 261.663,Z 407.838,A -85,B 0,C 180,E1 -19744.958,E2 -19744.958} C_VEL
LIN {X 0,Y 263.24,Z 400.916,A -85,B 0,C 180,E1 -19745.758,E2 -19745.758} C_VEL
LIN {X 0,Y 262.223,Z 394.353,A -85,B 0,C 180,E1 -19746.853,E2 -19746.853} C_VEL
LIN {X 0,Y 258.91,Z 381.873,A -85,B 0,C 180,E1 -19748.98,E2 -19748.98} C_VEL
LIN {X 0,Y 254.775,Z 370.173,A -85,B 0,C 180,E1 -19750.945,E2 -19750.945} C_VEL
LIN {X 0,Y 249.632,Z 358.564,A -85,B 0,C 180,E1 -19752.946,E2 -19752.946} C_VEL
